FUNCTION "PressureAi" : VOID	// FC 29
TITLE = Block for pressure analog input
//Building:
//Date         Editor                                                     Version
//--------------------------------------------------------------------------------
//10.05.2017   (gea)                                                      01.00.00
//
//Modifications:
//No. Date     Edit  Description                                    Index Version
//--------------------------------------------------------------------------------
//01  
//________________________________________________________________________________
//Functional description:
//
//The Pressure Analogue Input Object includes the following functions
//- Check of overflow with substitude value
//- scaling of input value
//- check of pressure levels
//- mode selection 
//  manual mode (empty / convey / overpressure | zero pint adjustment)
//- overpressure detection (with delay)
//- overpressure alarm (with delay)
//- empty pressure detection (with delay)
//- active pressure detection 
//- adjustment of zeropoint (autoamtic / manual)
//- data structure for HMI connection
//
AUTHOR : gea
VERSION : 1.0
VAR_INPUT
  ManOpEn : BOOL ;	// Enable Manual mode
  ManModeTrack : BOOL ;	// Manual mode PV tracking
  NegEvalEn : BOOL ;	// overpressure=0; underpressure=1
  OVErrEn : BOOL ;	// overflow/underflow/broken wire error enable
  AlarmOprEn : BOOL ;	// Alarm high enable
  AlarmOprAckEn : BOOL ;	// Alarm high acknowledge enable
  DigitMin : INT ;	// scaling digit max
  DigitMax : INT ;	// scaling digit min
  ValueMin : REAL ;	// scaling value max
  ValueMax : REAL ;	// scaling value min
  ValueSubs : REAL ;	// substitude value
  Configuration : WORD ;	// external Configuration (0=use internal)
  UOM : INT ;	// external Uom  (0=use internal)
  iSystemOn : BOOL ;	// System activated
  iwDigit : INT ;	// input digit value
  iActive : BOOL ;	// Pressure montioring active
  aAlarmOprAck : BOOL ;	// Alarm high acknowledge
END_VAR
VAR_IN_OUT
  PVAct : REAL ;
  fAlarmOpr : BOOL ;
  OverPressure : BOOL ;
  EmptyPressure : BOOL ;
  ActivePressure : BOOL ;
  fScalingErr : BOOL ;
  fOVErr : BOOL ;
  fParErr : BOOL ;
  ioStructure : ANY ;
END_VAR
VAR_TEMP
  State : INT ;
  tempReal1 : REAL ;
  tempReal2 : REAL ;
  tempDB : INT ;
  PVActRaw : REAL ;
  ScaleingErrPV : BOOL ;
  ScaleingErrOffset : BOOL ;
END_VAR
BEGIN
NETWORK
TITLE =  get start byte of structure
      L     P##ioStructure;
      LAR2;
      L     W [AR2,P#4.0];
      T     #tempDB;
      OPN   DI [#tempDB];
      L     D [AR2,P#6.0];
      LAR2;
NETWORK
TITLE =  external  configuration
      L     #Configuration;
      L     0;
      ==I;
      JC    NECO;
      L     #Configuration;
      L     0;
      <>I;
      =     DIX [AR2,P#0.0];	// PressureAinOn
      L     #Configuration;
      L     2#1000;
      AW;
      L     0;
      <>I;
      =     DIX [AR2,P#0.3];	// counter overpressure on
      L     #Configuration;
      L     2#10000;
      AW;
      L     0;
      <>I;
      =     DIX [AR2,P#0.4];	// counter emptypressure on
      L     #Configuration;
      L     2#100000;
      AW;
      L     0;
      <>I;
      =     DIX [AR2,P#0.5];	// counter activepressure on
      L     #Configuration;
      L     2#100000000;
      AW;
      L     0;
      <>I;
      =     DIX [AR2,P#1.0];	// overpressure parameter on
      L     #Configuration;
      L     2#1000000000;
      AW;
      L     0;
      <>I;
      =     DIX [AR2,P#1.1];	// emptypressure parameter on
      L     #Configuration;
      L     2#10000000000;
      AW;
      L     0;
      <>I;
      =     DIX [AR2,P#1.2];	// activeypressure parameter on
      L     #Configuration;
      L     2#1000000000000;
      AW;
      L     0;
      <>I;
      =     DIX [AR2,P#1.4];	// manual operation simulation on
      L     #Configuration;
      L     2#10000000000000;
      AW;
      L     0;
      <>I;
      =     DIX [AR2,P#1.5];	// manual operation adjust on
NECO: NOP   0;
      L     #UOM;
      L     0;
      ==I;
      JC    NEUO;
      L     #UOM;
      T     DIW [AR2,P#2.0];
NEUO: NOP   0;
NETWORK
TITLE =  clean up configuration
      O     DIX [AR2,P#0.3];	// counter overpressure on
      R     DIX [AR2,P#0.4];	// counter emptypressure on
      O     DIX [AR2,P#0.3];	// counter overpressure on
      O     DIX [AR2,P#0.4];	// counter emptypressure on
      R     DIX [AR2,P#0.5];	// counter activepressure on
NETWORK
TITLE =  selection manual mode
      A     DIX [AR2,P#4.1];	// ManModeOp
      AN    DIX [AR2,P#4.2];	// ManModeLock
      AN    "M0.0 LockManualMode";	// manual mode general disabled
      S     DIX [AR2,P#4.0];	// ManModAct
      ON    DIX [AR2,P#4.1];	// ManModeOp
      ON    #ManOpEn;	// manual mode local disabled
      O     "M0.0 LockManualMode";	// manual mode general disabled
      O     DIX [AR2,P#4.2];	// ManModeLock
      R     DIX [AR2,P#4.0];	// ManModAct
      R     DIX [AR2,P#4.1];	// ManModeOp
NETWORK
TITLE =  overflow / underflow / broken wire check
      O(;
      L     #iwDigit;
      L     32511;
      >I;
      );	//overflow
      O(;
      A(;
      L     #iwDigit;
      L     -32512;
      <I;
      );
      A(;
      L     #DigitMin;
      L     0;
      <>I;	//bipolar
      );
      );	//underflow bipolar
      O(;
      A(;
      L     #iwDigit;
      L     -4864;
      <I;
      );
      A(;
      L     #DigitMin;
      L     0;
      ==I;	//unipolar
      );
      );	//underflow //unipolar
      A     #OVErrEn;	//enable overflow / underflow error
      =     #fOVErr;
NETWORK
TITLE =  scaling of PV
//Val = ValueMin + (ValueMax-ValueMin)*(iwDigit-DigitMin)/(DigitMax-DigitMin)
// (network holds code this reader does not know; not shown)
NETWORK
TITLE =  substidue PV
      O     #fScalingErr;
      O     #fOVErr;
      AN    DIX [AR2,P#4.0];	// ManModAct
      JCN   PVSU;
      L     #ValueSubs;
      T     #PVAct;
PVSU: NOP   0;
NETWORK
TITLE =  manual mode PV: off
      A     DIX [AR2,P#4.0];	// ManModAct
      AN    DIX [AR2,P#4.3];	// ManOpPressureEmpty
      AN    DIX [AR2,P#4.4];	// ManOpPressureConveying
      AN    DIX [AR2,P#4.5];	// ManOpPressureAlarm
      A     DIX [AR2,P#1.4];	// ManOpSimEn
      JCN   PVMO;
      L     0.000000e+00;
      T     #PVAct;
PVMO: NOP   0;
NETWORK
TITLE =  manual mode PV: Emptypressure
      A     DIX [AR2,P#4.0];	// ManModAct
      A     DIX [AR2,P#4.3];	// ManOpPressureEmpty
      AN    DIX [AR2,P#4.4];	// ManOpPressureConveying
      AN    DIX [AR2,P#4.5];	// ManOpPressureAlarm
      A     DIX [AR2,P#1.4];	// ManOpSimEn
      JCN   PVME;
      L     DID [AR2,P#24.0];	//EmptypressurePV     
      L     DID [AR2,P#28.0];	//ActivePressurePV    
      -R;
      L     2.000000e+00;
      /R;
      L     DID [AR2,P#28.0];	//ActivePressurePV    
      +R;
      T     #PVAct;
PVME: NOP   0;
NETWORK
TITLE =  manual mode PV: convey pressure
      A     DIX [AR2,P#4.0];	// ManModAct
      A     DIX [AR2,P#4.4];	// ManOpPressureConveying
      AN    DIX [AR2,P#4.5];	// ManOpPressureAlarm
      A     DIX [AR2,P#1.4];	// ManOpSimEn
      JCN   PVMC;
      L     DID [AR2,P#16.0];	//MaxpressurePV     
      L     DID [AR2,P#24.0];	//EmptypressurePV     
      -R;
      L     2.000000e+00;
      /R;
      L     DID [AR2,P#24.0];	//EmptypressurePV     
      +R;
      T     #PVAct;
PVMC: NOP   0;
NETWORK
TITLE =  manual mode PV: overpressure
      A     DIX [AR2,P#4.0];	// ManModAct
      A     DIX [AR2,P#4.5];	// ManOpPressureAlarm
      A     DIX [AR2,P#1.4];	// ManOpSimEn
      JCN   PVMA;
      L     DID [AR2,P#16.0];	//MaxpressurePV     
      T     #PVAct;
PVMA: NOP   0;
NETWORK
TITLE =  check Parameter
// (network holds code this reader does not know; not shown)
NETWORK
TITLE =  overpressure detection
      A(;
      L     #PVAct;
      L     DID [AR2,P#16.0];	//MaxpressurePV     
      >=R;
      );
      AN    #NegEvalEn;
      A     #iActive;
      O;
      A(;
      L     #PVAct;
      L     DID [AR2,P#16.0];	//MaxpressurePV     
      <=R;
      );
      A     #NegEvalEn;
      A     #iActive;
      S     #OverPressure;
      A(;
      L     #PVAct;
      L     DID [AR2,P#20.0];	//MinpressurePV 
      <=R;
      );
      AN    #NegEvalEn;
      O;
      A(;
      L     #PVAct;
      L     DID [AR2,P#20.0];	//MinpressurePV 
      >=R;
      );
      A     #NegEvalEn;
      ON    #iActive;
      R     #OverPressure;
NETWORK
TITLE =  emptypressure detection
      A(;
      L     #PVAct;
      L     DID [AR2,P#24.0];	//EmptypressurePV     
      <=R;
      );
      AN    #NegEvalEn;
      A     #iActive;
      O;
      A(;
      L     #PVAct;
      L     DID [AR2,P#24.0];	//EmptypressurePV     
      >=R;
      );
      A     #NegEvalEn;
      A     #iActive;
      JCN   EPDC;
      A     "M4.5 ImpulseClock1,0Sec";
      AN    #EmptyPressure;
      L     DIW [AR2,P#38.0];	// EmptyDelayCounter
      JCN   EPDR;
      +     1;
      JU    EPDR;
EPDC: L     0;
EPDR: T     DIW [AR2,P#38.0];	// EmptyDelayCounter
      L     DIW [AR2,P#32.0];	// EmptyDelay
      >=I;
      =     #EmptyPressure;
NETWORK
TITLE =  activepressure detection
      A(;
      L     #PVAct;
      L     DID [AR2,P#28.0];	//ActivePressurePV    
      >=R;
      );
      A     #iActive;
      AN    #NegEvalEn;
      O;
      A(;
      L     #PVAct;
      L     DID [AR2,P#28.0];	//ActivePressurePV    
      <=R;
      );
      A     #iActive;
      A     #NegEvalEn;
      JCN   APDC;
      A     "M4.5 ImpulseClock1,0Sec";
      AN    #ActivePressure;
      L     DIW [AR2,P#40.0];	// ActiveDelayCounter
      JCN   APDR;
      +     1;
      JU    APDR;
APDC: L     0;
APDR: T     DIW [AR2,P#40.0];	// ActiveDelayCounter
      L     DIW [AR2,P#34.0];	// ActiveDelay
      >=I;
      =     #ActivePressure;
NETWORK
TITLE =  Alarm overpressure
      A     #OverPressure;
      A     #AlarmOprEn;
      A     #iActive;
      JCN   OPDC;
      A     "M4.5 ImpulseClock1,0Sec";
      AN    #fAlarmOpr;
      L     DIW [AR2,P#42.0];	// AlarmDelayCounter
      JCN   OPDR;
      +     1;
      JU    OPDR;
OPDC: L     0;
OPDR: T     DIW [AR2,P#42.0];	// AlarmDelayCounter
      L     DIW [AR2,P#36.0];	// AlarmDelay
      >=I;
      S     #fAlarmOpr;
      AN    #OverPressure;
      A(;
      A     #AlarmOprAckEn;
      A     #aAlarmOprAck;
      ON    #AlarmOprAckEn;
      );
      ON    #AlarmOprEn;
      ON    #iSystemOn;
      ON    #iActive;
      R     #fAlarmOpr;
NETWORK
TITLE =  adjust automatic
// (network holds code this reader does not know; not shown)
NETWORK
TITLE =  adjust manual
      AN    DIX [AR2,P#4.0];	// ManModeAct
      A     DIX [AR2,P#1.5];	// parameter.MapOpAdjustEn
      A     DIX [AR2,P#4.6];	// ManOpPressureAdjust
      =     DIX [AR2,P#6.4];	// ManAdjustReq
      A     DIX [AR2,P#1.5];	// parameter.MapOpAdjustEn
      A     DIX [AR2,P#4.6];	// ManOpPressureAdjust
      AN    #iActive;
      A     DIX [AR2,P#6.4];	// ManAdjustReq
      A     DIX [AR2,P#6.5];	// ManAdjustRdy
      JCN   ADMA;
      L     #PVActRaw;
      T     DID [AR2,P#12.0];	//PressureOffset
      SET;	// done!
      R     DIX [AR2,P#4.6];	// ManOpPressureAdjust
ADMA: NOP   0;
      ON    DIX [AR2,P#1.5];	// parameter.MapOpAdjustEn
      R     DIX [AR2,P#4.6];	// ManOpPressureAdjust
NETWORK
TITLE =  Switch counter count up
      A     #OverPressure;
      A     DIX [AR2,P#0.3];	// parameter.counterOverPressure
      O;
      A     #EmptyPressure;
      A     DIX [AR2,P#0.4];	// parameter.counterEmptyPressure
      O;
      A     #ActivePressure;
      A     DIX [AR2,P#0.5];	// parameter.counterActivePressure
      FP    DIX [AR2,P#6.7];	// Switch counter edge
      JCN   SCUP;
      L     1.000000e+00;
      L     DID [AR2,P#44.0];	// Switch counter
      +R;
      T     DID [AR2,P#44.0];	// Switch counter
SCUP: NOP   0;
NETWORK
TITLE =  Switch counter reset
      A     DIX [AR2,P#6.6];	// Switch counter Reset
      O;
      AN    DIX [AR2,P#0.3];	// parameter.counterOverPressure
      AN    DIX [AR2,P#0.5];	// parameter.counterEmptyPressure
      AN    DIX [AR2,P#0.4];	// parameter.counterActivePressure
      JCN   SCRE;
      R     DIX [AR2,P#6.6];	// Switch counter Reset
      L     0.000000e+00;
      T     DID [AR2,P#44.0];	// Switch counter
SCRE: NOP   0;
NETWORK
TITLE =  track manual mode value in automatic
      AN    DIX [AR2,P#4.0];	// ManModAct
      A     #ManModeTrack;
      AN    #fParErr;
      JCN   PVTK;
      AN    #ActivePressure;
      AN    #EmptyPressure;
      AN    #OverPressure;
      R     DIX [AR2,P#4.3];	// ManOpPressureEmpty
      R     DIX [AR2,P#4.4];	// ManOpPressureConveying
      R     DIX [AR2,P#4.5];	// ManOpPressureAlarm
      A     #ActivePressure;
      A     #EmptyPressure;
      AN    #OverPressure;
      S     DIX [AR2,P#4.3];	// ManOpPressureEmpty
      R     DIX [AR2,P#4.4];	// ManOpPressureConveying
      R     DIX [AR2,P#4.5];	// ManOpPressureAlarm
      A     #ActivePressure;
      AN    #EmptyPressure;
      AN    #OverPressure;
      R     DIX [AR2,P#4.3];	// ManOpPressureEmpty
      S     DIX [AR2,P#4.4];	// ManOpPressureConveying
      R     DIX [AR2,P#4.5];	// ManOpPressureAlarm
      A     #ActivePressure;
      AN    #EmptyPressure;
      A     #OverPressure;
      R     DIX [AR2,P#4.3];	// ManOpPressureEmpty
      R     DIX [AR2,P#4.4];	// ManOpPressureConveying
      S     DIX [AR2,P#4.5];	// ManOpPressureAlarm
PVTK: NOP   0;
NETWORK
TITLE =  Objektstatus für Visualisation OP (009) (010)
// 9 = scaling/overflow/underflow/broken wire: substitude value ==> grey 
      L     9;
      O     #fScalingErr;
      O     #fOVErr;
      JC    disp;
// 19 = system not on (interlock) ==> orange
      L     19;
      AN    #iSystemOn;
      JC    disp;
// 16 = alarm overpressure ==> red
      L     16;
      A     #fAlarmOpr;
      JC    disp;
// 16 = overpressure ==> yellow
      L     13;
      A     #OverPressure;
      AN    #fAlarmOpr;
      JC    disp;
// 5 = switch on ==> green
      L     5;
      A     #ActivePressure;
      AN    #EmptyPressure;
      JC    disp;
// 1 = switch off ==> cyan
      L     1;
      A     #ActivePressure;
      A     #EmptyPressure;
      JC    disp;
      L     0;
disp: T     #State;
NETWORK
TITLE =  save data to structure
      A     #iSystemOn;
      =     DIX [AR2,P#4.7];
      A     #fScalingErr;
      =     DIX [AR2,P#5.0];
      A     #fOVErr;
      =     DIX [AR2,P#5.1];
      A     #fParErr;
      =     DIX [AR2,P#5.2];
      A     #fAlarmOpr;
      =     DIX [AR2,P#5.3];
      A     #AlarmOprEn;
      =     DIX [AR2,P#5.4];
      A     #aAlarmOprAck;
      =     DIX [AR2,P#5.5];
      A     #OverPressure;
      =     DIX [AR2,P#5.6];
      A     #EmptyPressure;
      =     DIX [AR2,P#5.7];
      A     #ActivePressure;
      =     DIX [AR2,P#6.0];
      A     #iActive;
      =     DIX [AR2,P#6.1];
      L     #PVAct;
      T     DID [AR2,P#8.0];
      L     #State;
      T     DIW [AR2,P#48.0];	// #Objektstatus  (Struktur) 
END_FUNCTION

FUNCTION "FC30 DB vorbelegen" : VOID	// FC 30
TITLE = Baustein vorbelegen
//Erstellung:
//Datum        Bearbeiter                                                 Version
//--------------------------------------------------------------------------------
//08.12.98     R.Schaffert (sra)                                          01.00.00
//
//Änderungen:
//Nr. Datum    Bearb Beschreibung                                   Marke Version
//--------------------------------------------------------------------------------
//01  13.04.00 sra   Fehlerbehebung (1 Byte zuviel belegt)                01.00.01
//02  25.08.00 sra   Fehlerbehebung Zeigerberechnung                      01.00.02
//
//________________________________________________________________________________
//Beschreibung:
//
//Diese Funktion beschreibt die angegebenen Worte eines Datenbausteins mit dem im 
//Parameter "Wert" eingetragenen Wert.
//
AUTHOR : sra
FAMILY : AZO
VERSION : 0.0
VAR_INPUT
  DB_Nr : INT ;	//Datenbausteinnummer
  DW_Anfang : INT ;	//Anfangs-Datenwort im Datenbaustein
  Anzahl_Bytes : INT ;	//Anzahl der Bytes die vorbelegt werden sollen
  Wert : INT ;	//Wert mit dem der Bereich vorbelegt werden soll
END_VAR
VAR_TEMP
  Datenbaustein : INT ;
  Ptr_aktuelles_Datenbyte : DWORD ;
  Ptr_Ende_Datenbyte : DWORD ;
END_VAR
BEGIN
NETWORK
TITLE = Anzahl Worte prüfen
      L     #Anzahl_Bytes;
      L     0;
      <=I;
      JC    Ende;
NETWORK
TITLE = Datenbaustein öffnen
      L     #DB_Nr;
      T     #Datenbaustein;
      OPN   DB [#Datenbaustein];
NETWORK
TITLE = Pointer belegen
      L     #DW_Anfang;
      SLD   3;
      T     #Ptr_aktuelles_Datenbyte;
      L     #Anzahl_Bytes;
      L     #DW_Anfang;
      +I;
      SLD   3;
      T     #Ptr_Ende_Datenbyte;
NETWORK
TITLE = Wert schreiben
Loop: NOP   0;
      L     #Wert;
      T     DBB [#Ptr_aktuelles_Datenbyte];
      L     #Ptr_aktuelles_Datenbyte;	// Wortadresse um 1 erhöhen
      L     P#1.0;
      +D;
      T     #Ptr_aktuelles_Datenbyte;
      L     #Ptr_Ende_Datenbyte;
      <D;
      JC    Loop;
Ende: NOP   0;
END_FUNCTION

FUNCTION "FC40 copy Obj-SST Master" : VOID	// FC 40
TITLE = SST an Slave
//Erstellung:
//Datum        Bearbeiter                                                 Version
//--------------------------------------------------------------------------------
//22.03.01     R.Schaffert (sra)                                          01.00.00
//
//Änderungen:
//Nr. Datum    Bearb Beschreibung                                   Marke Version
//--------------------------------------------------------------------------------
//01  16.08.01 sra   Fehlerbeseitigung  Daten löschen               (001) 01.00.01
//02  31.08.01 sra   Daten von Ziel auch löschen wenn Ziel-DB 0 ist (002) 01.00.02
//
//________________________________________________________________________________
//Beschreibung: 
//
//Der Baustein kopiert die Schnittstelle, die durch den ANY-Zeiger festgelegt 
//ist, 
//an einen "Slave". Sobald ein Bit in der Steuerbitleiste gesetzt ist reagiert 
//der 
//Slave und antwortet. Ist kein Bit in der Steuerbitleiste belegt, baut der Slave 
//die Schnittstelle ab und kann durch anderen Master belegt werden.
//!!Die Steuerbitleiste ist immer das letzte Wort in der Schnittstelle!!
//
//Anwendung z.B. bei Kommunikation mehrere Waage <-> mehrere Silo  
// 
//
AUTHOR : sra
FAMILY : AZO
VERSION : 0.0
VAR_INPUT
  i_Freigabe : BOOL ;	//Freigabe der Kopierfunktion
  i_Ziel_DB : INT ;	//Ziel-Datenbaustein
  i_Ziel_DW : INT ;	//Ziel-Datenwort im Ziel-Datenbaustein
  i_SST_von_Ziel : ANY ;	//ANY-Zeiger auf Schnittstellen von Slave
  i_SST_an_Ziel : ANY ;	//ANY-Zeiger auf Schnittstellen an Slave
END_VAR
VAR_OUTPUT
  Ziel_frei : BOOL ;	//"Slave" ist nicht durch anderen Master belegt,die Daten können umkopiert werden
END_VAR
VAR_TEMP
  Quell_DB : INT ;
  SST_an_Anfangs_DW : INT ;
  SST_an_Laenge : INT ;
  SST_von_Anfangs_DW : INT ;
  SST_von_Laenge : INT ;
  Ziel_DB : INT ;
  Zaehler : INT ;
  Fehler_Blockkopieren : INT ;
END_VAR
BEGIN
NETWORK
TITLE = ANY Zeiger "SST_von_Ziel" zerlegen
      L     P##i_SST_von_Ziel;
      LAR2;
      L     W [AR2,P#2.0];
      T     #SST_von_Laenge;
      L     D [AR2,P#6.0];
      L     DW#16#FFFFFF;
      AD;
      SRD   3;
      T     #SST_von_Anfangs_DW;
NETWORK
TITLE = ANY Zeiger "SST_an_Ziel" zerlegen
      L     P##i_SST_an_Ziel;
      LAR2;
      L     W [AR2,P#2.0];
      T     #SST_an_Laenge;
      L     W [AR2,P#4.0];
      T     #Quell_DB;
      L     D [AR2,P#6.0];
      L     DW#16#FFFFFF;
      AD;
      SRD   3;
      T     #SST_an_Anfangs_DW;
NETWORK
TITLE = Prüfen ob Ziel-DB <> 0
      L     #i_Ziel_DB;
      L     0;
      ==I;
      JC    DEL1;	// 002
NETWORK
TITLE = Prüfen ob Slave belegt ist
      L     #i_Ziel_DB;
      T     #Ziel_DB;
      OPN   DB [#Ziel_DB];
      L     #i_Ziel_DW;
      SLD   3;
      LAR2;
      O(;	// Slave bereits belegt ?
      L     DBW [AR2,P#0.0];
      L     #Quell_DB;
      ==I;
      );
      O(;	// Slave frei ?
      L     DBW [AR2,P#0.0];
      L     0;
      ==I;
      );
      =     #Ziel_frei;
NETWORK
TITLE = Daten von Ziel löschen
DEL1: OPN   DB [#Quell_DB];
      L     #SST_von_Anfangs_DW;
      SLD   3;
      LAR2;
      L     #SST_von_Laenge;
DEL2: T     #Zaehler;
      L     0;
      T     DBB [AR2,P#0.0];
      L     P#1.0;	// (001)
      +AR2;	// (001)
      L     #Zaehler;
      LOOP  DEL2;
      ON    #i_Freigabe;
      ON    #Ziel_frei;
      O(;	// (002)
      L     #i_Ziel_DB;	// (002)
      L     0;	// (002)
      ==I;	// (002)
      );	// (002)
      BEC;
NETWORK
TITLE = Daten an Slave kopieren
      L     #SST_an_Anfangs_DW;
      SLD   3;
      LAR2;
      L     #Quell_DB;
      T     DBW [AR2,P#0.0];
      L     #SST_von_Anfangs_DW;
      T     DBW [AR2,P#2.0];
      CALL  "FC5 Blocktransfer" (
           Quell_Typ                := B#16#44,
           Quell_DB                 := #Quell_DB,
           Quell_DW                 := #SST_an_Anfangs_DW,
           Ziel_Typ                 := B#16#44,
           Ziel_DB                  := #i_Ziel_DB,
           Ziel_DW                  := #i_Ziel_DW,
           Block_Laenge             := #SST_an_Laenge,
           outFehler                := #Fehler_Blockkopieren);
END_FUNCTION

FUNCTION "FC41 copy Obj-SST Slave" : VOID	// FC 41
TITLE = SST an Master
//Erstellung:
//Datum        Bearbeiter                                                 Version
//--------------------------------------------------------------------------------
//22.03.01     R.Schaffert (sra)                                          01.00.00
//
//Änderungen:
//Nr. Datum    Bearb Beschreibung                                   Marke Version
//--------------------------------------------------------------------------------
//01  00.00.00 xxx   xxx                                            ???   01.xx.xx
//
//________________________________________________________________________________
//Beschreibung: 
//
//Der Baustein kopiert die Schnittstelle, die durch den ANY-Zeiger festgelegt 
//ist, an einen "Master". Sobald ein Bit in der Steuerbitleiste gesetzt ist 
//reagiert der Slave und antwortet. Ist kein Bit in der Steuerbitleiste belegt, 
//baut der Slave die Schnittstelle ab und kann durch anderen Master belegt werden.
//!!Die Steuerbitleiste ist immer das letzte Wort in der Schnittstelle!!
//
//Anwendung z.B. bei Kommunikation mehrere Waage <-> mehrere Silo  
// 
//
//
AUTHOR : sra
FAMILY : AZO
VERSION : 0.0
VAR_INPUT
  i_SST_von_Ziel : ANY ;	//ANY-Zeiger auf Schnittstelle von Master
  i_SST_an_Ziel : ANY ;	//ANY-Zeiger auf Schnittstelle an Master
END_VAR
VAR_TEMP
  SST_an_Anfangs_DW : INT ;
  SST_an_Laenge : INT ;
  SST_von_Anfangs_DW : INT ;
  SST_von_Laenge : INT ;
  Ptr_SST_von_Anfangs_DW : DWORD ;
  Ptr_SST_von_Steuerbits : DWORD ;	//Steuerbits = Anfangs-DW + Länge -2
  Quell_DB : INT ;
  Ziel_DB : INT ;
  Ziel_DW : INT ;
  Fehler_Blockkopieren : INT ;
END_VAR
BEGIN
NETWORK
TITLE = ANY Zeiger "SST_von_Ziel" zerlegen
      L     P##i_SST_von_Ziel;
      LAR2;
      L     W [AR2,P#2.0];	// Länge der Struktur
      T     #SST_von_Laenge;
      L     D [AR2,P#6.0];	// Anfangs-DW der Struktur
      L     DW#16#FFFFFF;
      AD;
      SRD   3;
      T     #SST_von_Anfangs_DW;
NETWORK
TITLE = ANY Zeiger "SST_an_Ziel" zerlegen
      L     P##i_SST_an_Ziel;
      LAR2;
      L     W [AR2,P#2.0];
      T     #SST_an_Laenge;
      L     W [AR2,P#4.0];
      T     #Quell_DB;
      L     D [AR2,P#6.0];
      L     DW#16#FFFFFF;
      AD;
      SRD   3;
      T     #SST_an_Anfangs_DW;
NETWORK
TITLE = Pointer bilden
      L     #SST_von_Anfangs_DW;
      SLD   3;
      T     #Ptr_SST_von_Anfangs_DW;
      L     #SST_von_Anfangs_DW;
      L     #SST_von_Laenge;
      +I;
      L     2;
      -I;
      SLD   3;
      T     #Ptr_SST_von_Steuerbits;
NETWORK
TITLE = Prüfen ob Anforderung vorhanden
      OPN   DB [#Quell_DB];
      O(;
      L     DBW [#Ptr_SST_von_Anfangs_DW];	// Ziel-DB
      L     0;
      ==I;
      );
      O(;
      L     DBW [#Ptr_SST_von_Steuerbits];	// Steuerbits
      L     0;
      ==I;
      );
      JC    DEL;
NETWORK
TITLE = Daten an Master kopieren
      LAR2  #Ptr_SST_von_Anfangs_DW;
      L     DBW [AR2,P#0.0];	// Ziel-DB aus Struktur "SST_von" ermitteln
      T     #Ziel_DB;
      L     DBW [AR2,P#2.0];	// Ziel-DW aus Struktur "SST_von" ermitteln
      T     #Ziel_DW;
      CALL  "FC5 Blocktransfer" (
           Quell_Typ                := B#16#44,
           Quell_DB                 := #Quell_DB,
           Quell_DW                 := #SST_an_Anfangs_DW,
           Ziel_Typ                 := B#16#44,
           Ziel_DB                  := #Ziel_DB,
           Ziel_DW                  := #Ziel_DW,
           Block_Laenge             := #SST_an_Laenge,
           outFehler                := #Fehler_Blockkopieren);
NETWORK
TITLE = Daten von Master löschen
DEL:  L     DBW [#Ptr_SST_von_Steuerbits];
      L     0;
      <>I;
      JC    DELS;
      L     0;
      T     DBW [#Ptr_SST_von_Anfangs_DW];
DELS: L     0;
      T     DBW [#Ptr_SST_von_Steuerbits];
END_FUNCTION

FUNCTION "FC47 Tabelle schreiben" : VOID	// FC 47
TITLE = Tabelle schreiben
//DATUM     BEARBEITER                                                    VERSION
//--------------------------------------------------------------------------------
//29.02.00  A. Geiger (gea)                                               01.00.00
//  
//Änderungen:
//Nr. Datum    Bearb Beschreibung                                   Marke Version
//--------------------------------------------------------------------------------
//01  30.08.00 gea   Neue Konzeption (Kopieren über Schleife)             02.00.00
//
//________________________________________________________________________________
//Beschreibung: 
//Datensatz in Tabelle schreiben
//
//Aufbau Tabelle:
//  Tabellen-DB: 
//               DBB0    ... DBB(n-1)  1.Zeile
//               DBB(n)  ... DBB(2n-1) 2.Zeile
//               DBB(2n) ... DBB(3n-1) 3.Zeile
//               usw.
//
//Die Anzahl der Spalten pro Zeile (n) ist abhängig von der Länge der "Quelle".
//Die "Quelle" muß ein ANY-Zeiger auf Bytes oder Stuct sein.
//eine Überprüfung auf Existenz und Länge des Tabellen-DBs wird durchgeführt.
//
AUTHOR : gea
FAMILY : AZO
VERSION : 0.0
VAR_INPUT
  in_Tabelle_DB : INT ;	//Tabellen-DB-Nr.
  in_Offset_DW : INT ;	//Offset erster Tabelleneintrag in Tabellen-DB
  in_Zeile_schreiben : INT ;	//Eintrag in Tabelle, der geschrieben werden soll
END_VAR
VAR_OUTPUT
  out_Fehler : INT ;	//Fehlerauswertung
END_VAR
VAR_IN_OUT
  io_Quelle : ANY ;	//Zeiger auf Quelldaten Block
END_VAR
VAR_TEMP
  G_DB_SAVE : INT ;	//Global-DB-Register
  I_DB_SAVE : INT ;	//Instanz-DB-Register
  Zeiger_Quelle : DWORD ;
  DB_Quelle : INT ;
  Zeiger_Ziel : DWORD ;
  DB_Ziel : INT ;
  Blocklaenge : INT ;
  Datentyp : BYTE ;
  Start_DBB : INT ;
END_VAR
BEGIN
NETWORK
TITLE = DB-Register sichern
      L     DBNO;
      T     #G_DB_SAVE;
      L     DINO;
      T     #I_DB_SAVE;
NETWORK
TITLE = ANY-Zeiger Quelle zerlegen
      L     P##io_Quelle;
      LAR1;
      L     B [AR1,P#1.0];
      T     #Datentyp;
      L     W [AR1,P#2.0];
      T     #Blocklaenge;
      L     W [AR1,P#4.0];
      T     #DB_Quelle;
      L     D [AR1,P#6.0];
      T     #Zeiger_Quelle;
NETWORK
TITLE = Blocklänge prüfen
      L     #Blocklaenge;
      L     0;
      <=I;
      JC    BLFE;	//Blocklänge Fehler
NETWORK
TITLE = Datentyp prüfen
      L     #Datentyp;
      L     2;	//Datentyp = Byte oder Struct
      ==I;
      JCN   DTFE;
NETWORK
TITLE = Start-DBB des gewählten Eintrags
      L     #in_Zeile_schreiben;
      L     1;
      -I;
      L     #Blocklaenge;
      *I;
      L     #in_Offset_DW;
      +I;
      T     #Start_DBB;	//Start des n-ten Eintrags
NETWORK
TITLE = Bereichszeiger Zielzeiger
      L     W#16#85;
      CAD;
      L     #Start_DBB;
      SLD   3;
      +D;
      T     #Zeiger_Ziel;
NETWORK
TITLE = Ziel-DB
      L     #in_Tabelle_DB;
      T     #DB_Ziel;
NETWORK
TITLE = DBs aufschlagen
      L     #DB_Quelle;
      L     0;
      <>I;
      JCN   QNDB;
      OPN   DB [#DB_Quelle];
      L     DBNO;
      L     0;
      <=I;
      JC    DBNX;	//Fehler DB existiert nicht
      L     #Zeiger_Quelle;
      SRW   3;	//Anfangsbyte
      L     #Blocklaenge;
      +I;
      L     DBLG;
      >I;
      JC    DBLF;	//Fehler DB Länge nicht ausreichend
      L     #Zeiger_Quelle;
      L     DW#16#FFFFFF;
      AD;
      L     W#16#84;
      CAD;
      +D;
      T     #Zeiger_Quelle;
QNDB: L     #DB_Ziel;
      L     0;
      <>I;
      JCN   ZNDB;
      OPN   DI [#DB_Ziel];
      L     DINO;
      L     0;
      <=I;
      JC    DBNX;	//Fehler DB existiert nicht
      L     #Start_DBB;
      L     #Blocklaenge;
      +I;
      L     DILG;
      >I;
      JC    DBLF;	//Fehler DB Länge nicht ausreichend
ZNDB: NOP   0;
NETWORK
TITLE = Bytes kopieren
//geschwindigkeitsopitmiert:
//- Schleifenzäehler bleibt in AKKU1 und AKKU2
//- Kopieren über Worte, letztes Byte (ungerade Bytezahl) separat.
// (network holds code this reader does not know; not shown)
NETWORK
TITLE = Fehlerauswertung
      L     0;	//kein Fehler
      JU    SEFE;	//  setze Fehlerausgang
      L     -1;	//Bereichszeiger Quelle falsch
      JU    SEFE;	//  setze Fehlerausgang
      L     -2;	//Bereichszeiger Ziel falsch
      JU    SEFE;	//  setze Fehlerausgang
BLFE: L     -3;	//Blocklänge falsch
      JU    SEFE;	//  setze Fehlerausgang
DBNX: L     -4;	//Datenbaustein nicht existent 
      JU    SEFE;	//  setze Fehlerausgang
DBLF: L     -5;	//Datenbaustein Längenfehler
      JU    SEFE;	//  setze Fehlerausgang
DTFE: L     -6;	//Fehler Datentyp in ANY-Zeiger
SEFE: T     #out_Fehler;
NETWORK
TITLE = DB-Register wiederherstellen
      OPN   DB [#G_DB_SAVE];
      OPN   DI [#I_DB_SAVE];
NETWORK
TITLE = BIE-Bit zuweisen
      L     #out_Fehler;
      L     0;
      ==I;
      SAVE;
END_FUNCTION

FUNCTION "FC104 Blocktransf. ANY-Z" : VOID	// FC 104
TITLE = BlockTransfer mit ANY-Zeiger als Ziel
//DATUM     BEARBEITER                                                    VERSION
//--------------------------------------------------------------------------------
//29.02.00  A. Geiger (gea)                                               01.00.00
//  
//Änderungen:
//Nr. Datum    Bearb Beschreibung                    Änderung       Marke Version
//--------------------------------------------------------------------------------
//01  06.07.00 gea   Neue Konzeption (Kopieren über Schleife)             02.00.00
//02  26.10.01 gea   Fehlerbehebung DB überprüfen                   (002) 02.00.01
//03  05.11.03 gea   Alle Datentypen zulassen                       (003) 02.00.02
//04  10.06.10 sra   Bereich > 32767 kopieren                       (004) 02.00.03
//________________________________________________________________________________
//
//Funktion:
//
//Beschreibung: Kopieren Quelle nach Ziel (ANY-Zeiger)
//
//Datentyp:
//  P - Peripherie
//  E - Eingänge
//  A - Ausgänge
//  M - Merker
//  D - Datenbaustein in Quell_DB bzw. Ziel_DB
//  I - Instanz-DB in DI-Register
//  G - Global-DB in DB-Register
//  L - Lokaldaten
//  K - Bausteinvorbelegen mit Konstante in Quell_DW (Low-Byte) (nur für Quelle)
//
//
//
//
//
//
//
//
//
//
//
//
//
//THE HORROR CONTINUES ...
AUTHOR : gea
VERSION : 0.0
VAR_INPUT
  in_Quell_Typ : CHAR ;
  in_Quell_DB : INT ;	//Ziel-DB bei DW-Transfer
  in_Quell_DW : INT ;	//Byte-Adresse der Quelle
  in_Ziel : ANY ;
END_VAR
VAR_OUTPUT
  out_Fehler : INT ;	//Fehlermeldung
END_VAR
VAR_TEMP
  G_DB_SAVE : INT ;	//Global-DB-Register
  I_DB_SAVE : INT ;	//Instanz-DB-Register
  Zeiger_Quelle : DWORD ;
  DB_Quelle : INT ;
  Zeiger_Ziel : DWORD ;
  DB_Ziel : INT ;
  Blocklaenge : INT ;
  Datentyp : BYTE ;
END_VAR
BEGIN
NETWORK
TITLE = DB-Register sichern
      L     DBNO;
      T     #G_DB_SAVE;
      L     DINO;
      T     #I_DB_SAVE;
NETWORK
TITLE = ANY-Zeiger Ziel zerlegen
      L     P##in_Ziel;
      LAR1;
      L     B [AR1,P#1.0];
      T     #Datentyp;
      L     W [AR1,P#2.0];
      T     #Blocklaenge;
      L     W [AR1,P#4.0];
      T     #DB_Ziel;
      L     D [AR1,P#6.0];
      T     #Zeiger_Ziel;
NETWORK
TITLE = Blocklänge prüfen
      L     #Blocklaenge;
      L     0;
      <=I;
      JC    BLFE;	//Blocklänge Fehler
NETWORK
TITLE = Datentyp prüfen
      L     #Datentyp;
      L     0;	//Datentyp = Byte oder Struct //(003)
      <>I;
      JCN   DTFE;
NETWORK
TITLE = Bereichskennung Quellzeiger
      L     #in_Quell_Typ;
      L     'P';
      ==I;
      L     W#16#80;
      JC    BEKQ;
      L     #in_Quell_Typ;
      L     'E';
      ==I;
      L     W#16#81;
      JC    BEKQ;
      L     #in_Quell_Typ;
      L     'A';
      ==I;
      L     W#16#82;
      JC    BEKQ;
      L     #in_Quell_Typ;
      L     'M';
      ==I;
      L     W#16#83;
      JC    BEKQ;
      L     #in_Quell_Typ;
      L     'D';
      ==I;
      L     W#16#84;
      JC    BEKQ;
      L     #in_Quell_Typ;
      L     'I';
      ==I;
      L     W#16#84;
      JC    BEKQ;
      L     #in_Quell_Typ;
      L     'G';
      ==I;
      L     W#16#84;
      JC    BEKQ;
      L     #in_Quell_Typ;
      L     'L';
      ==I;
      L     W#16#87;
      JC    BEKQ;
      L     #in_Quell_Typ;
      L     'K';
      ==I;
      L     L#0;
      JC    BEK1;
      JU    BEFQ;	//Bereichskennung falsch Quelle
BEKQ: CAD;
      L     #in_Quell_DW;
      SLD   3;
      +D;
BEK1: T     #Zeiger_Quelle;
NETWORK
TITLE = Quell-DB
      L     #in_Quell_Typ;
      L     'D';
      ==I;
      L     #in_Quell_DB;
      JC    DBQ;
      L     #in_Quell_Typ;
      L     'I';
      ==I;
      L     DINO;
      JC    DBQ;
      L     #in_Quell_Typ;
      L     'G';
      ==I;
      L     DBNO;
      JC    DBQ;
      L     0;
DBQ:  T     #DB_Quelle;
NETWORK
TITLE = DBs aufschlagen
      O(;	//(002)
      L     #in_Quell_Typ;	//(002)
      L     'D';	//(002)
      ==I;	//(002)
      );	//(002)
      O(;	//(002)
      L     #in_Quell_Typ;	//(002)
      L     'I';	//(002)
      ==I;	//(002)
      );	//(002)
      O(;	//(002)
      L     #in_Quell_Typ;	//(002)
      L     'G';	//(002)
      ==I;	//(002)
      );	//(002)
      JCN   QNDB;
      OPN   DB [#DB_Quelle];
      L     DBNO;
      L     0;
      <=I;
      JC    DBNX;	//Fehler DB existiert nicht
      L     #in_Quell_DW;
      L     #Blocklaenge;
      +D;	// (004)
      L     DBLG;
      >D;	// (004)
      JC    DBLF;	//Fehler DB Länge nicht ausreichend
QNDB: L     #DB_Ziel;
      L     0;
      <>I;
      JCN   ZNDB;
      OPN   DI [#DB_Ziel];
      L     DINO;
      L     0;
      <=I;
      JC    DBNX;	//Fehler DB existiert nicht
      L     #Zeiger_Ziel;
      SRW   3;	//Anfangsbyte
      L     #Blocklaenge;
      +D;	// (004)
      L     DILG;
      >D;	// (004)
      JC    DBLF;	//Fehler DB Länge nicht ausreichend
      L     #Zeiger_Ziel;
      L     DW#16#FFFFFF;
      AD;
      L     W#16#85;
      CAD;
      +D;
      T     #Zeiger_Ziel;
ZNDB: NOP   0;
NETWORK
TITLE = Bereich vorbelegen
//geschwindigkeitsopitmiert:
//- Schleifenzäehler bleibt in AKKU1 und AKKU2
//- Kopieren über Worte, letztes Byte (ungerade Bytezahl) separat.
      L     #in_Quell_Typ;
      L     'K';
      ==I;
      JCN   NKCO;
      L     #Zeiger_Ziel;
      LAR2;
      L     #in_Quell_DW;	//Konstante für vorbelegen
      L     #in_Quell_DW;
      SLW   8;	//  In AKKU1LL und AKKU1LH
      OW;
      L     #Blocklaenge;	//Schleifenzähler Blocklaenge->AKKU1
      SRW   1;
SCHK: TAK;	//Schleifenzähler AKKU1->AKKU2; Vorbelegwert in AKKU1
      T     W [AR2,P#0.0];
      +AR2  P#2.0;
      TAK;	//Schleifenzähler in AKKU2->AKKU1; Vorbelegwert in AKKU2
      LOOP  SCHK;
      JZ    BLGK;	//Gerade Byteanzahl A1=0 und A0=0 nach "SRW 1"
      L     #in_Quell_DW;	//Ungerade Bytezahl letztes Byte einzeln Kopieren
      SRW   8;
      T     B [AR2,P#0.0];
BLGK: NOP   0;
      JU    BLGE;
NKCO: NOP   0;
NETWORK
TITLE = Bytes kopieren
//geschwindigkeitsopitmiert:
//- Schleifenzäehler bleibt in AKKU1 und AKKU2
//- Kopieren über Worte, letztes Byte (ungerade Bytezahl) separat.
// (network holds code this reader does not know; not shown)
NETWORK
TITLE = Fehlerauswertung
      L     0;	//kein Fehler
      JU    SEFE;	//  setze Fehlerausgang
BEFQ: L     -1;	//Bereichszeiger Quelle falsch
      JU    SEFE;	//  setze Fehlerausgang
      L     -2;	//Bereichszeiger Ziel falsch
      JU    SEFE;	//  setze Fehlerausgang
BLFE: L     -3;	//Blocklänge falsch
      JU    SEFE;	//  setze Fehlerausgang
DBNX: L     -4;	//Datenbaustein nicht existent 
      JU    SEFE;	//  setze Fehlerausgang
DBLF: L     -5;	//Datenbaustein Längenfehler
      JU    SEFE;	//  setze Fehlerausgang
DTFE: L     -6;	//Fehler Datentyp in ANY-Zeiger
SEFE: T     #out_Fehler;
NETWORK
TITLE = DB-Register wiederherstellen
      OPN   DB [#G_DB_SAVE];
      OPN   DI [#I_DB_SAVE];
NETWORK
TITLE = BIE-Bit zuweisen
      L     #out_Fehler;
      L     0;
      ==I;
      SAVE;
END_FUNCTION

FUNCTION "FC113 Standardsignale 2" : VOID	// FC 113
TITLE = function for several cabinets with their own fuse check
//Erstellung:
//Date        developer                                                  version
//--------------------------------------------------------------------------------
//18.07.2016  A.Kremer (kal)                                             01.00.00
//
//changes:
//No. Date    developer description                                 Mark  version
//--------------------------------------------------------------------------------
//
//________________________________________________________________________________
//function:
//function, if more than one cabinet handle their own fuse check.
//function can be called several times, then.
//
AUTHOR : kal
FAMILY : AZO
VERSION : 0.0
VAR_INPUT
  iFaultFuse_OK : BOOL ;	//Eingang Sicherung OK = Eingang Störung Sicherung
END_VAR
VAR_OUTPUT
  qlFaultFuse : BOOL ;	//Ausgang der Lampe "Störung Sicherung"
  qFaultFuse : BOOL ;	//Störung Sicherung -> für Störbitzuweisung im DB34
END_VAR
BEGIN
NETWORK
TITLE = lamp "fault fuse" and fault message
      AN    #iFaultFuse_OK;
      =     #qlFaultFuse;
      =     #qFaultFuse;
END_FUNCTION

FUNCTION "FC6079 SimAnalog" : INT	// FC 6079
TITLE = simulate analog signal
//creation:
//date         who                                                         version
//--------------------------------------------------------------------------------
//28.12.2010   M. Junker (jm)                                             01.00.00
//
//changes:
//no. date       who            what                                       version
//--------------------------------------------------------------------------------
// 1  
//
//Function:
//simulates a slow changing analog signal (pressure, temperature) for 
//visualization tests or program tests
//
//y = a * sin(x) + b
AUTHOR : jm
FAMILY : AZO
NAME : SIMUL
VERSION : 0.1
VAR_INPUT
  RELEASE : BOOL ;	//release simulation
  PERIOD : REAL ;	//period time for sin() [s]
  MAX : REAL ;	//maximum analog value to simulate
  MIN : REAL ;	//minimum analog value to simulate
  DEFAULT : REAL ;	//default value if not simulating
  MAXVALUE : REAL ;	//upper limit analog value
  MINVALUE : REAL ;	//lower limit analog value
END_VAR
VAR_OUTPUT
  RET_VAL : INT ;	//simulated analog signal
END_VAR
VAR_IN_OUT
  STARTTIME : TIME ;	//starttime [ms]
  ONESHOTSTART : BOOL ;	//help flag start
END_VAR
VAR_TEMP
  ACTTIME : TIME ;
  y : REAL ;
  x : REAL ;
  a : REAL ;
  b : REAL ;
  MR1 : REAL ;
  MR2 : REAL ;
END_VAR
BEGIN
NETWORK
TITLE = detect start time
      A     #RELEASE;
      FP    #ONESHOTSTART;
      JCN   NSST;	// Not Set Start Time
      CALL  "TIME_TCK" (
           RET_VAL                  := #STARTTIME);
NSST: NOP   0;
NETWORK
TITLE = check if simulation necessary
      A     #RELEASE;
      JC    CONT;
      L     #DEFAULT;
      T     #y;
      JU    OUT;	// scale value for output
NETWORK
TITLE = calculate x
//x = 2*pi/1000/PERIOD*deltaTms = deltaTms*pi/500/PERIOD
CONT: CALL  "TIME_TCK" (
           RET_VAL                  := #ACTTIME);
      L     #ACTTIME;
      L     #STARTTIME;
      -D;	// deltaT in ms 
      DTR;
      L     3.141593e+00;	// PI
      *R;
      L     5.000000e+02;
      /R;
      L     #PERIOD;
      /R;
      T     #x;
NETWORK
TITLE = calculate a
//a = (MAX-MIN)/2
      L     #MAX;
      L     #MIN;
      -R;
      L     2.000000e+00;
      /R;
      T     #a;
NETWORK
TITLE = calculate b
//b = (MAX+MIN)/2
      L     #MAX;
      L     #MIN;
      +R;
      L     2.000000e+00;
      /R;
      T     #b;
NETWORK
TITLE = calculate y
//y = a*sin(x)+b
// (network holds code this reader does not know; not shown)
NETWORK
TITLE = scale output
//z = (MAXDIGIT-MINDIGIT)/(MAXVALUE-MINVALUE)*(y-MINVALUE)+MINDIGIT 
OUT:  L     #MAXVALUE;
      L     #MINVALUE;
      -R;
      T     #MR1;
      L     #y;
      L     #MINVALUE;
      -R;
      T     #MR2;
      L     2.764800e+04;
      L     #MR1;
      /R;
      L     #MR2;
      *R;
      RND;
      T     #RET_VAL;
END_FUNCTION

FUNCTION "FC6091 SimValve3A3E" : VOID	// FC 6091
TITLE = simulate valve 3A3E
//creation:
//date         who                                                         version
//--------------------------------------------------------------------------------
//04.12.2015   M. Junker (jm)                                             01.00.00
//
//changes:
//no. date       who            what                                       version
//--------------------------------------------------------------------------------
// 1  
//
//Function:
//simulate valve
AUTHOR : jm
FAMILY : AZO
NAME : SIMUL
VERSION : 1.0
VAR_INPUT
  o_ValveOn : BOOL ;
  o_ValveOff : BOOL ;
  o_ValveSealup : BOOL ;
END_VAR
VAR_OUTPUT
  i_ValveOn : BOOL ;	//on, open, pos1, ...
  i_ValveOff : BOOL ;	//off, closed, pos2, ...
  i_ValveSealed : BOOL ;	//sealed
END_VAR
VAR_IN_OUT
  mPosition : BOOL ;	//help memory
END_VAR
BEGIN
NETWORK
TITLE = valve on
      A     #o_ValveOn;
      S     #mPosition;
NETWORK
TITLE = valve off
      A     #o_ValveOff;
      R     #mPosition;
NETWORK
TITLE = indications
      A     #mPosition;
      =     #i_ValveOn;
      NOT;
      =     #i_ValveOff;
NETWORK
TITLE = sealed
      A     #o_ValveSealup;
      =     #i_ValveSealed;
END_FUNCTION

FUNCTION "FC6092 SimValveDOS" : VOID	// FC 6092
TITLE = simulate valve 2A2E (dosing valve)
//creation:
//date         who                                                         version
//--------------------------------------------------------------------------------
//05.06.2014   M. Junker (jm)                                             01.00.00
//
//changes:
//no. date       who            what                                       version
//--------------------------------------------------------------------------------
// 1  
//
//Function:
//simulate valve
AUTHOR : jm
FAMILY : AZO
NAME : SIMUL
VERSION : 1.0
VAR_INPUT
  in_Ventil_Typ : INT ;	//siehe Funktionsbeschreibung unten
  o_ValveCoarse : BOOL ;
  o_ValveFine : BOOL ;
END_VAR
VAR_OUTPUT
  i_ValveOpen : BOOL ;	//on, open, pos1, ...
  i_ValveClosed : BOOL ;	//off, closed, pos2, ...
END_VAR
VAR_IN_OUT
  mPosition : BOOL ;	//help memory
END_VAR
BEGIN
NETWORK
TITLE = valve open
      A     #o_ValveCoarse;
      S     #mPosition;
NETWORK
TITLE = valve  closed
      AN    #o_ValveCoarse;
      AN    #o_ValveFine;
      R     #mPosition;
NETWORK
TITLE = valve type 0
      A(;
      L     #in_Ventil_Typ;
      L     0;
      );
      <>I;
      JC    NVT0;
      A     #o_ValveCoarse;
      =     #i_ValveOpen;
      AN    #o_ValveCoarse;
      AN    #o_ValveFine;
      =     #i_ValveClosed;
NVT0: NOP   0;
NETWORK
TITLE = valve type 1
      A(;
      L     #in_Ventil_Typ;
      L     1;
      );
      <>I;
      JC    NVT1;
      A     #mPosition;
      =     #i_ValveOpen;
      AN    #mPosition;
      =     #i_ValveClosed;
NVT1: NOP   0;
NETWORK
TITLE = valve type 2
      A(;
      L     #in_Ventil_Typ;
      L     2;
      );
      <>I;
      JC    NVT2;
      A     #mPosition;
      =     #i_ValveOpen;
      AN    #mPosition;
      =     #i_ValveClosed;
NVT2: NOP   0;
END_FUNCTION

FUNCTION "FC6093 SimValveDS" : VOID	// FC 6093
TITLE = simulate valve 2A2E (double seat)
//creation:
//date         who                                                         version
//--------------------------------------------------------------------------------
//27.05.2014   M. Junker (jm)                                             01.00.00
//
//changes:
//no. date       who            what                                       version
//--------------------------------------------------------------------------------
// 1  
//
//Function:
//simulate valve
AUTHOR : jm
FAMILY : AZO
NAME : SIMUL
VERSION : 1.0
VAR_INPUT
  o_Valve_E0 : BOOL ;
  o_Valve_E1 : BOOL ;
END_VAR
VAR_OUTPUT
  i_Valve_A0 : BOOL ;	//on, open, pos1, ...
  i_Valve_A1 : BOOL ;	//off, closed, pos2, ...
END_VAR
BEGIN
NETWORK
TITLE = valve open
      A     #o_Valve_E0;
      A     #o_Valve_E1;
      =     #i_Valve_A1;
NETWORK
TITLE = valve close
      ON    #o_Valve_E0;
      ON    #o_Valve_E1;
      =     #i_Valve_A0;
END_FUNCTION

FUNCTION "FC6094 SimMotor2A2E" : VOID	// FC 6094
TITLE = simulate motor 2A2E+iso
//creation:
//date         who                                                         version
//--------------------------------------------------------------------------------
//05.06.2014   M. Junker (jm)                                             01.00.00
//
//changes:
//no. date       who            what                                       version
//--------------------------------------------------------------------------------
// 1  
//
//Function:
//simulate motor + isolator
AUTHOR : jm
FAMILY : AZO
NAME : SIMUL
VERSION : 1.0
VAR_INPUT
  o_MotorCW : BOOL ;
  o_MotorACW : BOOL ;
  Isolators : BOOL ;
END_VAR
VAR_OUTPUT
  i_MotorCW : BOOL ;
  i_MotorACW : BOOL ;
  i_IsoMotor : BOOL ;
END_VAR
BEGIN
NETWORK
TITLE = motor CW
      A     #o_MotorCW;
      =     #i_MotorCW;
NETWORK
TITLE = motor ACW
      A     #o_MotorACW;
      =     #i_MotorACW;
NETWORK
TITLE = isolator
      A     #Isolators;
      =     #i_IsoMotor;
END_FUNCTION

FUNCTION "FC6095 SimValve2A2E" : VOID	// FC 6095
TITLE = simulate valve 2A2E
//creation:
//date         who                                                         version
//--------------------------------------------------------------------------------
//25.10.2010   M. Junker (jm)                                             01.00.00
//
//changes:
//no. date       who            what                                       version
//--------------------------------------------------------------------------------
// 1  
//
//Function:
//simulate valve
AUTHOR : jm
FAMILY : AZO
NAME : SIMUL
VERSION : 1.0
VAR_INPUT
  o_ValveOn : BOOL ;
  o_ValveOff : BOOL ;
END_VAR
VAR_OUTPUT
  i_ValveOn : BOOL ;	//on, open, pos1, ...
  i_ValveOff : BOOL ;	//off, closed, pos2, ...
END_VAR
VAR_IN_OUT
  mPosition : BOOL ;	//help memory
END_VAR
BEGIN
NETWORK
TITLE = valve on
      A     #o_ValveOn;
      S     #mPosition;
NETWORK
TITLE = valve off
      A     #o_ValveOff;
      R     #mPosition;
NETWORK
TITLE = indications
      A     #mPosition;
      =     #i_ValveOn;
      NOT;
      =     #i_ValveOff;
END_FUNCTION

FUNCTION "FC6096 SimValve1AE1" : VOID	// FC 6096
TITLE = simulate valve 1AE1
//creation:
//date         who                                                         version
//--------------------------------------------------------------------------------
//25.10.2010   M. Junker (jm)                                             01.00.00
//
//changes:
//no. date       who            what                                       version
//--------------------------------------------------------------------------------
// 1  
//
//Function:
//simulate valve
AUTHOR : jm
FAMILY : AZO
NAME : SIMUL
VERSION : 1.0
VAR_INPUT
  o_ValveOn : BOOL ;
END_VAR
VAR_OUTPUT
  i_ValveOff : BOOL ;	//off, closed, pos2, ...
END_VAR
BEGIN
NETWORK
TITLE = valve off
      AN    #o_ValveOn;
      =     #i_ValveOff;
END_FUNCTION

FUNCTION "FC6097 SimValve1A1E" : VOID	// FC 6097
TITLE = simulate valve 1A1E
//creation:
//date         who                                                         version
//--------------------------------------------------------------------------------
//25.10.2010   M. Junker (jm)                                             01.00.00
//
//changes:
//no. date       who            what                                       version
//--------------------------------------------------------------------------------
// 1  
//
//Function:
//simulate valve
AUTHOR : jm
FAMILY : AZO
NAME : SIMUL
VERSION : 1.0
VAR_INPUT
  o_ValveOn : BOOL ;
END_VAR
VAR_OUTPUT
  i_ValveOn : BOOL ;	//on, open, pos1, ...
END_VAR
BEGIN
NETWORK
TITLE = valve on
      A     #o_ValveOn;
      =     #i_ValveOn;
END_FUNCTION

FUNCTION "FC6098 SimValve1A2E" : VOID	// FC 6098
TITLE = simulate valve 1A2E
//creation:
//date         who                                                         version
//--------------------------------------------------------------------------------
//25.10.2010   M. Junker (jm)                                             01.00.00
//
//changes:
//no. date       who            what                                       version
//--------------------------------------------------------------------------------
// 1  
//
//Function:
//simulate valve
AUTHOR : jm
FAMILY : AZO
NAME : SIMUL
VERSION : 1.0
VAR_INPUT
  o_ValveOn : BOOL ;
END_VAR
VAR_OUTPUT
  i_ValveOn : BOOL ;	//on, open, pos1, ...
  i_ValveOff : BOOL ;	//off, closed, pos2, ...
END_VAR
BEGIN
NETWORK
TITLE = valve on
      A     #o_ValveOn;
      =     #i_ValveOn;
NETWORK
TITLE = valve off
      AN    #o_ValveOn;
      =     #i_ValveOff;
END_FUNCTION

FUNCTION "FC6099 SimMotor1A1E" : VOID	// FC 6099
TITLE = simulate motor 1A1E+iso
//creation:
//date         who                                                         version
//--------------------------------------------------------------------------------
//25.10.2010   M. Junker (jm)                                             01.00.00
//
//changes:
//no. date       who            what                                       version
//--------------------------------------------------------------------------------
// 1  
//
//Function:
//simulate motor + isolator
AUTHOR : jm
FAMILY : AZO
NAME : SIMUL
VERSION : 1.0
VAR_INPUT
  o_MotorOn : BOOL ;
  Isolators : BOOL ;
END_VAR
VAR_OUTPUT
  i_MotorOn : BOOL ;
  i_IsoMotor : BOOL ;
END_VAR
BEGIN
NETWORK
TITLE = motor
      A     #o_MotorOn;
      =     #i_MotorOn;
NETWORK
TITLE = isolator
      A     #Isolators;
      =     #i_IsoMotor;
END_FUNCTION

DATA_BLOCK "CMs_SIMULATION_DB"	// DB 2
VERSION : 0.0
"CMs_SIMULATION"
BEGIN
END_DATA_BLOCK

DATA_BLOCK "DB3 CPU Daten"	// DB 3
AUTHOR : sra
FAMILY : AZO
VERSION : 0.0
  STRUCT
   OB1_Info : STRUCT
    OB1_DATE_TIME : DATE_AND_TIME ;	//Date and time OB1 started
    OB1_PREV_CYCLE : INT ;	//Cycle time of previous OB1 scan (milliseconds)
    OB1_MIN_CYCLE : INT ;	//Minimum cycle time of OB1 (milliseconds)
    OB1_MAX_CYCLE : INT ;	//Maximum cycle time of OB1 (milliseconds)
    reserve : ARRAY  [0 .. 14 ] OF BYTE ;
   END_STRUCT ;
   Fehler_OB_Info : STRUCT
    Zeitfehler_OB80 : BOOL ;	//Zeitfehler OB 80
    Stromversorgung_OB81 : BOOL ;	//Stromversorgungsfehler OB 81
    Diagnose_Alarm_OB82 : BOOL ;	//Diagnose-Alarm OB82
    Ziehen_Stecken_OB83 : BOOL ;	//Ziehen/Stecken-Alarm OB83
    CPU_Hardware_OB84 : BOOL ;	//CPU-Hardwarefehler OB84
    Programmablauf_OB85 : BOOL ;	//Programmablauffehler OB85
    Baugr_tr_ausfall_OB86 : BOOL ;	//Baugruppenträgerausfall OB86
    Kommunikation_OB87 : BOOL ;	//Kommunikationsfehler OB87
    Programmierfehler_OB121 : BOOL ;	//Programmierfehler OB121
    Periphzugriff_OB122 : BOOL ;	//Peripheriezugriffsfehler OB 122
    Bearbeitungsabbruch_OB88 : BOOL ;	//Bearbeitungsabbruch eines Bausteins OB88
    Battery_fault : BOOL ;	//Battery fault with SFC51
    reserve_word : WORD ;
    OB_80_Fault_ID : BYTE ;	//Fehlercode OB 80
    OB_81_Fault_ID : BYTE ;	//Fehlercode OB 81
    OB_82_Fault_ID : BYTE ;	//Fehlercode OB 82
    OB_83_Fault_ID : BYTE ;	//Fehlercode OB 83
    OB_84_Fault_ID : BYTE ;	//Fehlercode OB 84
    OB_85_Fault_ID : BYTE ;	//Fehlercode OB 85
    OB_86_Fault_ID : BYTE ;	//Fehlercode OB 86
    OB_87_Fault_ID : BYTE ;	//Fehlercode OB 87
    OB_121_Fault_ID : BYTE ;	//Fehlercode OB 121
    OB_122_Fault_ID : BYTE ;	//Fehlercode OB 122
    OB_88_Fault_ID : BYTE ;	//Fehlercode OB 122
    reserve : ARRAY  [16 .. 29 ] OF BYTE ;
   END_STRUCT ;
   RDSYSST : STRUCT
    BUSY : BOOL ;
    RETVAL : INT ;
    SLZ_HEADER : STRUCT
     LENTHDR : WORD ;
     N_DR : WORD ;
    END_STRUCT ;
    DR : STRUCT
     Data_1 : BYTE ;
     Data_2 : BYTE ;
     Data_3 : BYTE ;
     Data_4 : BYTE ;
     Data_5 : BYTE ;
     Data_6 : BYTE ;
     Data_7 : BYTE ;
     Data_8 : BYTE ;
     Data_9 : BYTE ;
     Data_10 : BYTE ;
     Data_11 : BYTE ;
     Data_12 : BYTE ;
     Data_13 : BYTE ;
     Data_14 : BYTE ;
     Data_15 : BYTE ;
     Data_16 : BYTE ;
     Data_17 : BYTE ;
     Data_18 : BYTE ;
     Data_19 : BYTE ;
     Data_20 : BYTE ;
    END_STRUCT ;
   END_STRUCT ;
  END_STRUCT ;	
BEGIN
END_DATA_BLOCK

DATA_BLOCK "DB4 Motordaten für FUs"	// DB 4
VERSION : 0.1
  STRUCT
   Motordaten1 : STRUCT 	//Anzahl der Motordaten abhängig von der Anzahl der verschied. benutzten Motoren
    Nennleistungsfaktor : REAL  := 8.000000e-001;	//Motornennleistungsfaktor cos phi
    Nennfrequenz : REAL  := 5.100000e+001;	//Motornennfrequenz in Einheit Hz
    Nenndrehzahl : REAL  := 1.400000e+003;	//Motornenndrehzal in U/min
    Nennstrom : REAL  := 6.100000e+000;	//Motornennstrom in A
    Nennspannung : REAL  := 2.310000e+002;	//Motornennspannung in V
    Nennleistung : REAL  := 1.400000e+000;	//Motornennleistung kW
    reserve : ARRAY  [24 .. 29 ] OF //Reserve für weitere Motordaten
    BYTE ;
   END_STRUCT ;
   Motordaten2 : STRUCT
    Nennleistungsfaktor : REAL  := 7.000000e-001;
    Nennfrequenz : REAL  := 1.000000e+002;
    Nenndrehzahl : REAL  := 2.000000e+002;
    Nennstrom : REAL  := 2.000000e+000;
    Nennspannung : REAL  := 3.800000e+002;
    Nennleistung : REAL  := 1.000000e+003;
    reserve : ARRAY  [24 .. 29 ] OF BYTE ;
   END_STRUCT ;
   Motordaten3 : STRUCT
    Nennleistungsfaktor : REAL  := 7.000000e-001;
    Nennfrequenz : REAL  := 1.000000e+002;
    Nenndrehzahl : REAL  := 2.000000e+002;
    Nennstrom : REAL  := 5.000000e+000;
    Nennspannung : REAL  := 3.800000e+002;
    Nennleistung : REAL  := 1.000000e+003;
    reserve : ARRAY  [24 .. 29 ] OF BYTE ;
   END_STRUCT ;
   Motordaten4 : STRUCT
    Nennleistungsfaktor : REAL  := 7.000000e-001;
    Nennfrequenz : REAL  := 1.000000e+002;
    Nenndrehzahl : REAL  := 2.000000e+002;
    Nennstrom : REAL  := 5.000000e+000;
    Nennspannung : REAL  := 3.800000e+002;
    Nennleistung : REAL  := 1.000000e+003;
    reserve : ARRAY  [24 .. 29 ] OF BYTE ;
   END_STRUCT ;
   Motordaten5 : STRUCT
    Nennleistungsfaktor : REAL  := 7.000000e-001;
    Nennfrequenz : REAL  := 1.000000e+002;
    Nenndrehzahl : REAL  := 2.000000e+002;
    Nennstrom : REAL  := 5.000000e+000;
    Nennspannung : REAL  := 3.800000e+002;
    Nennleistung : REAL  := 1.000000e+003;
    reserve : ARRAY  [24 .. 29 ] OF BYTE ;
   END_STRUCT ;
   Motordaten6 : STRUCT
    Nennleistungsfaktor : REAL  := 7.000000e-001;
    Nennfrequenz : REAL  := 1.000000e+002;
    Nenndrehzahl : REAL  := 2.000000e+002;
    Nennstrom : REAL  := 5.000000e+000;
    Nennspannung : REAL  := 3.800000e+002;
    Nennleistung : REAL  := 1.000000e+003;
    reserve : ARRAY  [24 .. 29 ] OF BYTE ;
   END_STRUCT ;
   Motordaten7 : STRUCT
    Nennleistungsfaktor : REAL  := 7.000000e-001;
    Nennfrequenz : REAL  := 1.000000e+002;
    Nenndrehzahl : REAL  := 2.000000e+002;
    Nennstrom : REAL  := 5.000000e+000;
    Nennspannung : REAL  := 3.800000e+002;
    Nennleistung : REAL  := 1.000000e+003;
    reserve : ARRAY  [24 .. 29 ] OF BYTE ;
   END_STRUCT ;
   Motordaten8 : STRUCT
    Nennleistungsfaktor : REAL  := 7.000000e-001;
    Nennfrequenz : REAL  := 1.000000e+002;
    Nenndrehzahl : REAL  := 2.000000e+002;
    Nennstrom : REAL  := 5.000000e+000;
    Nennspannung : REAL  := 3.800000e+002;
    Nennleistung : REAL  := 1.000000e+003;
    reserve : ARRAY  [24 .. 29 ] OF BYTE ;
   END_STRUCT ;
   Motordaten9 : STRUCT
    Nennleistungsfaktor : REAL  := 7.000000e-001;
    Nennfrequenz : REAL  := 1.000000e+002;
    Nenndrehzahl : REAL  := 2.000000e+002;
    Nennstrom : REAL  := 5.000000e+000;
    Nennspannung : REAL  := 3.800000e+002;
    Nennleistung : REAL  := 1.000000e+003;
    reserve : ARRAY  [24 .. 29 ] OF BYTE ;
   END_STRUCT ;
   Motordaten10 : STRUCT
    Nennleistungsfaktor : REAL  := 7.000000e-001;
    Nennfrequenz : REAL  := 1.000000e+002;
    Nenndrehzahl : REAL  := 2.000000e+002;
    Nennstrom : REAL  := 5.000000e+000;
    Nennspannung : REAL  := 3.800000e+002;
    Nennleistung : REAL  := 1.000000e+003;
    reserve : ARRAY  [24 .. 29 ] OF BYTE ;
   END_STRUCT ;
  END_STRUCT ;	
BEGIN
   Motordaten1.Nennleistungsfaktor := 8.000000e-01;
   Motordaten1.Nennfrequenz := 5.100000e+01;
   Motordaten1.Nenndrehzahl := 1.400000e+03;
   Motordaten1.Nennstrom := 6.100000e+00;
   Motordaten1.Nennspannung := 2.310000e+02;
   Motordaten1.Nennleistung := 1.400000e+00;
   Motordaten2.Nennleistungsfaktor := 7.000000e-01;
   Motordaten2.Nennfrequenz := 1.000000e+02;
   Motordaten2.Nenndrehzahl := 2.000000e+02;
   Motordaten2.Nennstrom := 5.000000e+00;
   Motordaten2.Nennspannung := 3.800000e+02;
   Motordaten2.Nennleistung := 1.000000e+03;
   Motordaten3.Nennleistungsfaktor := 7.000000e-01;
   Motordaten3.Nennfrequenz := 1.000000e+02;
   Motordaten3.Nenndrehzahl := 2.000000e+02;
   Motordaten3.Nennstrom := 5.000000e+00;
   Motordaten3.Nennspannung := 3.800000e+02;
   Motordaten3.Nennleistung := 1.000000e+03;
   Motordaten4.Nennleistungsfaktor := 7.000000e-01;
   Motordaten4.Nennfrequenz := 1.000000e+02;
   Motordaten4.Nenndrehzahl := 2.000000e+02;
   Motordaten4.Nennstrom := 5.000000e+00;
   Motordaten4.Nennspannung := 3.800000e+02;
   Motordaten4.Nennleistung := 1.000000e+03;
   Motordaten5.Nennleistungsfaktor := 7.000000e-01;
   Motordaten5.Nennfrequenz := 1.000000e+02;
   Motordaten5.Nenndrehzahl := 2.000000e+02;
   Motordaten5.Nennstrom := 5.000000e+00;
   Motordaten5.Nennspannung := 3.800000e+02;
   Motordaten5.Nennleistung := 1.000000e+03;
   Motordaten6.Nennleistungsfaktor := 7.000000e-01;
   Motordaten6.Nennfrequenz := 1.000000e+02;
   Motordaten6.Nenndrehzahl := 2.000000e+02;
   Motordaten6.Nennstrom := 5.000000e+00;
   Motordaten6.Nennspannung := 3.800000e+02;
   Motordaten6.Nennleistung := 1.000000e+03;
   Motordaten7.Nennleistungsfaktor := 7.000000e-01;
   Motordaten7.Nennfrequenz := 1.000000e+02;
   Motordaten7.Nenndrehzahl := 2.000000e+02;
   Motordaten7.Nennstrom := 5.000000e+00;
   Motordaten7.Nennspannung := 3.800000e+02;
   Motordaten7.Nennleistung := 1.000000e+03;
   Motordaten8.Nennleistungsfaktor := 7.000000e-01;
   Motordaten8.Nennfrequenz := 1.000000e+02;
   Motordaten8.Nenndrehzahl := 2.000000e+02;
   Motordaten8.Nennstrom := 5.000000e+00;
   Motordaten8.Nennspannung := 3.800000e+02;
   Motordaten8.Nennleistung := 1.000000e+03;
   Motordaten9.Nennleistungsfaktor := 7.000000e-01;
   Motordaten9.Nennfrequenz := 1.000000e+02;
   Motordaten9.Nenndrehzahl := 2.000000e+02;
   Motordaten9.Nennstrom := 5.000000e+00;
   Motordaten9.Nennspannung := 3.800000e+02;
   Motordaten9.Nennleistung := 1.000000e+03;
   Motordaten10.Nennleistungsfaktor := 7.000000e-01;
   Motordaten10.Nennfrequenz := 1.000000e+02;
   Motordaten10.Nenndrehzahl := 2.000000e+02;
   Motordaten10.Nennstrom := 5.000000e+00;
   Motordaten10.Nennspannung := 3.800000e+02;
   Motordaten10.Nennleistung := 1.000000e+03;
END_DATA_BLOCK

DATA_BLOCK "DB30 Daten von/an FG"	// DB 30
AUTHOR : sra
FAMILY : hsh
VERSION : 0.0
"FB30 Daten von/an  FG"
BEGIN
END_DATA_BLOCK

DATA_BLOCK "DB32 Inputs"	// DB 32
AUTHOR : sra
FAMILY : SCADA
VERSION : 0.0
"FB32 Eingaege an FG"
BEGIN
END_DATA_BLOCK

DATA_BLOCK "DB33 Outputs"	// DB 33
AUTHOR : sra
FAMILY : SCADA
VERSION : 0.0
"FB33 Ausgaege an FG"
BEGIN
END_DATA_BLOCK

DATA_BLOCK "DB34 Faults"	// DB 34
AUTHOR : sra
FAMILY : AZO
VERSION : 0.0
"FB34 Störbearbeitung"
BEGIN
END_DATA_BLOCK

DATA_BLOCK "DB35 Acknolegments"	// DB 35
VERSION : 0.1
  STRUCT
   Quittierung : ARRAY  [0 .. 1023, 0 .. 7 ] OF BOOL  := FALSE;
   Quittierung_Spiegelungen : ARRAY  [0 .. 1023, 0 .. 7 ] OF BOOL  := FALSE;
  END_STRUCT ;	
BEGIN
END_DATA_BLOCK

DATA_BLOCK "DB92 Eingänge AVP"	// DB 92
VERSION : 0.0
"FB92 Eingänge AVP"
BEGIN
END_DATA_BLOCK

DATA_BLOCK "LINE1"	// DB 1000
AUTHOR : ilia
VERSION : 0.0
"****PRODUCTION****"
BEGIN
END_DATA_BLOCK

DATA_BLOCK "CONTAINERSTATION CST01"	// DB 1001
AUTHOR : ilia
VERSION : 0.1
"CONTAINERSTATION"
BEGIN
END_DATA_BLOCK

DATA_BLOCK "RECEIVER REC01"	// DB 1011
AUTHOR : ilia
VERSION : 0.1
"RECEIVER"
BEGIN
END_DATA_BLOCK

DATA_BLOCK "VP01"	// DB 1051
AUTHOR : ilia
VERSION : 0.1
"VACUUM PUMP"
BEGIN
END_DATA_BLOCK

DATA_BLOCK "RecipeData"	// DB 1111
VERSION : 0.1
  STRUCT
   RECIPE1 : STRUCT 	//Recipe
    RecipeName : STRING  [18 ] := 'RECIPE1';	//Recipe Name
    SpeedRinne : INT  := 30;	//Speed of Rinne
    SpeedRotaryFeeder : INT  := 30;	//Speed of RF
    SpeedVacuumPump : INT  := 35;	//Speed of VP1
    NumberOfPumps : INT  := 1;
    reserve1 : INT ;
    reserve2 : INT ;
    reserve3 : ARRAY  [1 .. 8 ] OF BYTE  := B#16#0;
   END_STRUCT ;
   RECIPE2 : STRUCT 	//Recipe
    RecipeName : STRING  [18 ] := 'RECIPE2';	//Recipe Name
    SpeedRinne : INT  := 30;	//Speed of Rinne
    SpeedRotaryFeeder : INT  := 30;	//Speed of RF
    SpeedVacuumPump : INT  := 35;	//Speed of VP1
    NumberOfPumps : INT  := 1;
    reserve1 : INT ;
    reserve2 : INT ;
    reserve3 : ARRAY  [1 .. 8 ] OF BYTE  := B#16#0;
   END_STRUCT ;
   RECIPE3 : STRUCT 	//Recipe
    RecipeName : STRING  [18 ] := 'RECIPE3';	//Recipe Name
    SpeedRinne : INT  := 30;	//Speed of Rinne
    SpeedRotaryFeeder : INT  := 30;	//Speed of RF
    SpeedVacuumPump : INT  := 35;	//Speed of VP1
    NumberOfPumps : INT  := 1;
    reserve1 : INT ;
    reserve2 : INT ;
    reserve3 : ARRAY  [1 .. 8 ] OF BYTE  := B#16#0;
   END_STRUCT ;
   RECIPE4 : STRUCT 	//Recipe
    RecipeName : STRING  [18 ] := 'RECIPE4';	//Recipe Name
    SpeedRinne : INT  := 30;	//Speed of Rinne
    SpeedRotaryFeeder : INT  := 30;	//Speed of RF
    SpeedVacuumPump : INT  := 35;	//Speed of VP1
    NumberOfPumps : INT  := 1;
    reserve1 : INT ;
    reserve2 : INT ;
    reserve3 : ARRAY  [1 .. 8 ] OF BYTE  := B#16#0;
   END_STRUCT ;
   RECIPE5 : STRUCT 	//Recipe
    RecipeName : STRING  [18 ] := 'RECIPE5';	//Recipe Name
    SpeedRinne : INT  := 30;	//Speed of Rinne
    SpeedRotaryFeeder : INT  := 30;	//Speed of RF
    SpeedVacuumPump : INT  := 35;	//Speed of VP1
    NumberOfPumps : INT  := 1;
    reserve1 : INT ;
    reserve2 : INT ;
    reserve3 : ARRAY  [1 .. 8 ] OF BYTE  := B#16#0;
   END_STRUCT ;
   RECIPE6 : STRUCT 	//Recipe
    RecipeName : STRING  [18 ] := 'RECIPE6';	//Recipe Name
    SpeedRinne : INT  := 30;	//Speed of Rinne
    SpeedRotaryFeeder : INT  := 30;	//Speed of RF
    SpeedVacuumPump : INT  := 35;	//Speed of VP1
    NumberOfPumps : INT  := 1;
    reserve1 : INT ;
    reserve2 : INT ;
    reserve3 : ARRAY  [1 .. 8 ] OF BYTE  := B#16#0;
   END_STRUCT ;
   RECIPE7 : STRUCT 	//Recipe
    RecipeName : STRING  [18 ] := 'RECIPE7';	//Recipe Name
    SpeedRinne : INT  := 30;	//Speed of Rinne
    SpeedRotaryFeeder : INT  := 30;	//Speed of RF
    SpeedVacuumPump : INT  := 35;	//Speed of VP1
    NumberOfPumps : INT  := 1;
    reserve1 : INT ;
    reserve2 : INT ;
    reserve3 : ARRAY  [1 .. 8 ] OF BYTE  := B#16#0;
   END_STRUCT ;
   RECIPE8 : STRUCT 	//Recipe
    RecipeName : STRING  [18 ] := 'RECIPE8';	//Recipe Name
    SpeedRinne : INT  := 30;	//Speed of Rinne
    SpeedRotaryFeeder : INT  := 30;	//Speed of RF
    SpeedVacuumPump : INT  := 35;	//Speed of VP1
    NumberOfPumps : INT  := 1;
    reserve1 : INT ;
    reserve2 : INT ;
    reserve3 : ARRAY  [1 .. 8 ] OF BYTE  := B#16#0;
   END_STRUCT ;
   RECIPE9 : STRUCT 	//Recipe
    RecipeName1 : STRING  [18 ] := 'RECIPE9';	//Recipe Name
    SpeedRinne : INT  := 30;	//Speed of Rinne
    SpeedRotaryFeeder : INT  := 30;	//Speed of RF
    SpeedVacuumPump : INT  := 35;	//Speed of VP1
    NumberOfPumps : INT  := 1;
    reserve1 : INT ;
    reserve2 : INT ;
    reserve3 : ARRAY  [1 .. 8 ] OF BYTE  := B#16#0;
   END_STRUCT ;
   RECIPE10 : STRUCT 	//Recipe
    RecipeName : STRING  [18 ] := 'RECIPE10';	//Recipe Name
    SpeedRinne : INT  := 30;	//Speed of Rinne
    SpeedRotaryFeeder : INT  := 30;	//Speed of RF
    SpeedVacuumPump : INT  := 35;	//Speed of VP1
    NumberOfPumps : INT  := 1;
    reserve1 : INT ;
    reserve2 : INT ;
    reserve3 : ARRAY  [1 .. 8 ] OF BYTE  := B#16#0;
   END_STRUCT ;
  END_STRUCT ;	
BEGIN
   RECIPE1.RecipeName := 'RECIPE1';
   RECIPE1.SpeedRinne := 30;
   RECIPE1.SpeedRotaryFeeder := 30;
   RECIPE1.SpeedVacuumPump := 35;
   RECIPE1.NumberOfPumps := 1;
   RECIPE2.RecipeName := 'RECIPE2';
   RECIPE2.SpeedRinne := 30;
   RECIPE2.SpeedRotaryFeeder := 30;
   RECIPE2.SpeedVacuumPump := 35;
   RECIPE2.NumberOfPumps := 1;
   RECIPE3.RecipeName := 'RECIPE3';
   RECIPE3.SpeedRinne := 30;
   RECIPE3.SpeedRotaryFeeder := 30;
   RECIPE3.SpeedVacuumPump := 35;
   RECIPE3.NumberOfPumps := 1;
   RECIPE4.RecipeName := 'RECIPE4';
   RECIPE4.SpeedRinne := 30;
   RECIPE4.SpeedRotaryFeeder := 30;
   RECIPE4.SpeedVacuumPump := 35;
   RECIPE4.NumberOfPumps := 1;
   RECIPE5.RecipeName := 'RECIPE5';
   RECIPE5.SpeedRinne := 30;
   RECIPE5.SpeedRotaryFeeder := 30;
   RECIPE5.SpeedVacuumPump := 35;
   RECIPE5.NumberOfPumps := 1;
   RECIPE6.RecipeName := 'RECIPE6';
   RECIPE6.SpeedRinne := 30;
   RECIPE6.SpeedRotaryFeeder := 30;
   RECIPE6.SpeedVacuumPump := 35;
   RECIPE6.NumberOfPumps := 1;
   RECIPE7.RecipeName := 'RECIPE7';
   RECIPE7.SpeedRinne := 30;
   RECIPE7.SpeedRotaryFeeder := 30;
   RECIPE7.SpeedVacuumPump := 35;
   RECIPE7.NumberOfPumps := 1;
   RECIPE8.RecipeName := 'RECIPE8';
   RECIPE8.SpeedRinne := 30;
   RECIPE8.SpeedRotaryFeeder := 30;
   RECIPE8.SpeedVacuumPump := 35;
   RECIPE8.NumberOfPumps := 1;
   RECIPE9.RecipeName1 := 'RECIPE9';
   RECIPE9.SpeedRinne := 30;
   RECIPE9.SpeedRotaryFeeder := 30;
   RECIPE9.SpeedVacuumPump := 35;
   RECIPE9.NumberOfPumps := 1;
   RECIPE10.RecipeName := 'RECIPE10';
   RECIPE10.SpeedRinne := 30;
   RECIPE10.SpeedRotaryFeeder := 30;
   RECIPE10.SpeedVacuumPump := 35;
   RECIPE10.NumberOfPumps := 1;
END_DATA_BLOCK

DATA_BLOCK "test"	// DB 2222
VERSION : 0.1
  STRUCT
   Recipe : STRUCT 	//Temporary placeholder variable
    Speed_1 : INT  := 1;
    Speed_2 : INT  := 2;
    Number : INT ;
   END_STRUCT ;
  END_STRUCT ;	
BEGIN
   Recipe.Speed_1 := 1;
   Recipe.Speed_2 := 2;
END_DATA_BLOCK

DATA_BLOCK "FREQUENCY CONVERTERS"	// DB 4900
AUTHOR : ilia
VERSION : 0.0
"*** FCs ***"
BEGIN
END_DATA_BLOCK

DATA_BLOCK "FC VACUUM PUMP"	// DB 10001
VERSION : 0.0
"FREQ.CONVERTER"
BEGIN
END_DATA_BLOCK

DATA_BLOCK "FC ROTARY FEEDER REC01"	// DB 10002
VERSION : 0.0
"FREQ.CONVERTER"
BEGIN
END_DATA_BLOCK

ORGANIZATION_BLOCK "OB 1 Zyklisches Prg."	// OB 1
TITLE = zyklischer Programmablauf
//Erstellung:
//Datum        Bearbeiter                                                 Version
//--------------------------------------------------------------------------------
//01.08.18     Ilia Bedniakov                                             01.00.00
//
//Änderungen:
//Nr. Datum    Bearb Beschreibung                                   Marke Version
//--------------------------------------------------------------------------------
//01  
//
VERSION : 0.1
VAR_TEMP
  OB1_EV_CLASS : BYTE ;	//Bits 0-3 = 1 (Coming event), Bits 4-7 = 1 (Event class 1)
  OB1_SCAN_1 : BYTE ;	//1 (Cold restart scan 1 of OB 1), 3 (Scan 2-n of OB 1)
  OB1_PRIORITY : BYTE ;	//1 (Priority of 1 is lowest)
  OB1_OB_NUMBR : BYTE ;	//1 (Organization block 1, OB1)
  OB1_RESERVED_1 : BYTE ;	//Reserved for system
  OB1_RESERVED_2 : BYTE ;	//Reserved for system
  OB1_PREV_CYCLE : INT ;	//Cycle time of previous OB1 scan (milliseconds)
  OB1_MIN_CYCLE : INT ;	//Minimum cycle time of OB1 (milliseconds)
  OB1_MAX_CYCLE : INT ;	//Maximum cycle time of OB1 (milliseconds)
  OB1_DATE_TIME : DATE_AND_TIME ;	//Date and time OB1 started
  DUMMY_INT : INT ;
  dummybool : BOOL ;
END_VAR
BEGIN
NETWORK
TITLE = Simulation
//      CLR   
      SET;
      =     "M0.5 SimulationInternal";
      A     "M0.5 SimulationInternal";
      JCN   NS;	// No simulation
      CALL  "CMs_SIMULATION" , "CMs_SIMULATION_DB";
NS:   NOP   0;
NETWORK
TITLE = Datum, Uhrzeit und Zykluszeiten in DB3 kopieren
      CALL  "BLKMOV" (
           SRCBLK                   := #OB1_DATE_TIME,
           RET_VAL                  := #DUMMY_INT,
           DSTBLK                   := "DB3 CPU Daten".OB1_Info.OB1_DATE_TIME);
      L     #OB1_PREV_CYCLE;
      T     "DB3 CPU Daten".OB1_Info.OB1_PREV_CYCLE;
      L     #OB1_MIN_CYCLE;
      T     "DB3 CPU Daten".OB1_Info.OB1_MIN_CYCLE;
      L     #OB1_MAX_CYCLE;
      T     "DB3 CPU Daten".OB1_Info.OB1_MAX_CYCLE;
NETWORK
TITLE = Standardsignale
      CALL  "FC13 Standardsignale" (
           in_E_Sicherung_OK        := "01_01_101_Gn",
           in_Basistakt_Timer       := "M4.1 ImpulseClock0,2Sec",
           in_Zeit_Basistakt_100ms  := 2,
           o_Lampe_Stoer_Sicherung  := #dummybool,
           o_Stoerung_Sicherung     := #dummybool);
NETWORK
TITLE = Daten von/an HMI
      CALL  "FB30 Daten von/an  FG" , "DB30 Daten von/an FG";
      CALL  "FB32 Eingaege an FG" , "DB32 Inputs";
      CALL  "FB33 Ausgaege an FG" , "DB33 Outputs";
NETWORK
TITLE = Stoerungen Auswertung
      CALL  "FB34 Störbearbeitung" , "DB34 Faults";
NETWORK
TITLE = Anwenderprogramm
      CALL  "****PRODUCTION****" , "LINE1";
NETWORK
TITLE = Neustart oder Wiederanlauf SPS rücksetzen
//letztes Netzwerk
      SET;
      R     "M1.3 CompleteRestart";
      R     "M1.4 RestartPLC";
END_ORGANIZATION_BLOCK

ORGANIZATION_BLOCK "OB 80 Zeitfehler-OB"	// OB 80
TITLE = Zeitfehler
//Erstellung:
//Datum        Bearbeiter                                                 Version
//--------------------------------------------------------------------------------
//03.06.98     Rainer Schaffert (sra)                                     01.00.00
//
//Änderungen:
//Nr. Datum    Bearb Beschreibung                                   Marke Version
//--------------------------------------------------------------------------------
//01  
//
//________________________________________________________________________________
//OB wird bei Zeitfehler bearbeitet
//
AUTHOR : sra
FAMILY : error_OB
NAME : time_err
VERSION : 0.1
VAR_TEMP
  OB80_EV_CLASS : BYTE ;	//16#35, Event class 3, Entering event state, Internal fault event
  OB80_FLT_ID : BYTE ;	//16#XX, Fault identifcation code
  OB80_PRIORITY : BYTE ;	//26 (Priority of 1 is lowest)
  OB80_OB_NUMBR : BYTE ;	//80 (Organization block 80, OB80)
  OB80_RESERVED_1 : BYTE ;	//Reserved for system
  OB80_RESERVED_2 : BYTE ;	//Reserved for system
  OB80_ERROR_INFO : WORD ;	//Error information on event
  OB80_ERR_EV_CLASS : BYTE ;	//Class of event causing error
  OB80_ERR_EV_NUM : BYTE ;	//Number of event causing error
  OB80_OB_PRIORITY : BYTE ;	//Priority of OB causing error
  OB80_OB_NUM : BYTE ;	//Number of OB causing error
  OB80_DATE_TIME : DATE_AND_TIME ;	//Date and time OB80 started
END_VAR
BEGIN
NETWORK
TITLE = Fehlermeldung erzeugen
//Fehlermeldung erzeugen
//
//Fehlercode B#16#01 : Zykluszeit überschritten
//                     OB80_ERROR_INFO: Laufzeit des letzten Zyklus
//           
//           B#16#02 : Der angeforderte OB ist noch in Bearbeitung
//
//           B#16#07 : Überlauf des OB-Anforderungspuffers für die aktuelle 
//                     Prioritätsklasse
//
//           B#16#05 : abgelaufener Urzeitalarm durch Urzeitsprung
//
//           B#16#06 : abgelaufener Urzeitalarm bei Wiedereintritt 
//
      L     #OB80_FLT_ID;
      L     B#16#0;
      <>I;
      =     "DB3 CPU Daten".Fehler_OB_Info.Zeitfehler_OB80;
      L     #OB80_FLT_ID;
      T     "DB3 CPU Daten".Fehler_OB_Info.OB_80_Fault_ID;
END_ORGANIZATION_BLOCK

ORGANIZATION_BLOCK "OB 82 Diagnosealarm-OB"	// OB 82
TITLE = Diagnose-Alarm
//Erstellung:
//Datum        Bearbeiter                                                 Version
//--------------------------------------------------------------------------------
//03.06.98     Rainer Schaffert (sra)                                     01.00.00
//
//Änderungen:
//Nr. Datum    Bearb Beschreibung                                   Marke Version
//--------------------------------------------------------------------------------
//01  
//
//________________________________________________________________________________
//OB wird bei Diagnose-Alarm bearbeitet
//
AUTHOR : sra
FAMILY : error_OB
NAME : diagn_OB
VERSION : 0.1
VAR_TEMP
  OB82_EV_CLASS : BYTE ;	//16#39, Event class 3, Entering event state, Internal fault event
  OB82_FLT_ID : BYTE ;	//16#XX, Fault identifcation code
  OB82_PRIORITY : BYTE ;	//26/28 (Priority of 1 is lowest)
  OB82_OB_NUMBR : BYTE ;	//82 (Organization block 82, OB82)
  OB82_RESERVED_1 : BYTE ;	//Reserved for system
  OB82_IO_FLAG : BYTE ;	//Input (01010100), Output (01010101)
  OB82_MDL_ADDR : INT ;	//Base address of module with fault
  OB82_MDL_DEFECT : BOOL ;	//Module defective
  OB82_INT_FAULT : BOOL ;	//Internal fault
  OB82_EXT_FAULT : BOOL ;	//External fault
  OB82_PNT_INFO : BOOL ;	//Point information
  OB82_EXT_VOLTAGE : BOOL ;	//External voltage low
  OB82_FLD_CONNCTR : BOOL ;	//Field wiring connector missing
  OB82_NO_CONFIG : BOOL ;	//Module has no configuration data
  OB82_CONFIG_ERR : BOOL ;	//Module has configuration error
  OB82_MDL_TYPE : BYTE ;	//Type of module
  OB82_SUB_NDL_ERR : BOOL ;	//Sub-Module is missing or has error
  OB82_COMM_FAULT : BOOL ;	//Communication fault
  OB82_MDL_STOP : BOOL ;	//Module is stopped
  OB82_WTCH_DOG_FLT : BOOL ;	//Watch dog timer stopped module
  OB82_INT_PS_FLT : BOOL ;	//Internal power supply fault
  OB82_PRIM_BATT_FLT : BOOL ;	//Primary battery is in fault
  OB82_BCKUP_BATT_FLT : BOOL ;	//Backup battery is in fault
  OB82_RESERVED_2 : BOOL ;	//Reserved for system
  OB82_RACK_FLT : BOOL ;	//Rack fault, only for bus interface module
  OB82_PROC_FLT : BOOL ;	//Processor fault
  OB82_EPROM_FLT : BOOL ;	//EPROM fault
  OB82_RAM_FLT : BOOL ;	//RAM fault
  OB82_ADU_FLT : BOOL ;	//ADU fault
  OB82_FUSE_FLT : BOOL ;	//Fuse fault
  OB82_HW_INTR_FLT : BOOL ;	//Hardware interupt input in fault
  OB82_RESERVED_3 : BOOL ;	//Reserved for system
  OB82_DATE_TIME : DATE_AND_TIME ;	//Date and time OB82 started
END_VAR
BEGIN
NETWORK
TITLE = Fehlermeldung erzeugen
//Fehlermeldung erzeugen
//
//Fehlercode B#16#42 : 
//
      A(;
      L     #OB82_EV_CLASS;
      L     B#16#39;	// kommendes Ereignis
      ==I;
      );
      A(;
      L     #OB82_FLT_ID;
      L     B#16#0;
      <>I;
      );
      =     "DB3 CPU Daten".Fehler_OB_Info.Diagnose_Alarm_OB82;
      L     #OB82_FLT_ID;
      T     "DB3 CPU Daten".Fehler_OB_Info.OB_82_Fault_ID;
END_ORGANIZATION_BLOCK

ORGANIZATION_BLOCK "OB 83 Ziehen-/Stecken-OB"	// OB 83
TITLE = Ziehen/Stecken-Alarm
//Erstellung:
//Datum        Bearbeiter                                                 Version
//--------------------------------------------------------------------------------
//03.06.98     Rainer Schaffert (sra)                                     01.00.00
//
//Änderungen:
//Nr. Datum    Bearb Beschreibung                                   Marke Version
//--------------------------------------------------------------------------------
//01  
//
//________________________________________________________________________________
//OB wird bei Ziehen/Stecken-Alarm bearbeitet
//
AUTHOR : sra
FAMILY : AZO
VERSION : 0.0
VAR_TEMP
  OB83_EV_CLASS : BYTE ;	//16#38/39, Event class 3, module inserted/removed (8/9)
  OB83_FLT_ID : BYTE ;	//16#XX, Fault identifcation code
  OB83_PRIORITY : BYTE ;	//26/28 (Priority of 1 is lowest)
  OB83_OB_NUMBR : BYTE ;	//83 (Organization block 83, OB83)
  OB83_RESERVED_1 : BYTE ;	//Reserved for system
  OB83_MDL_ID : BYTE ;	//Input module (01010100), Output module (01010101)
  OB83_MDL_ADDR : WORD ;	//Base address of module with point fault
  OB83_RACK_NUM : WORD ;	//Number of rack that has module with point fault
  OB83_MDL_TYPE : WORD ;	//Module type with point fault
  OB83_DATE_TIME : DATE_AND_TIME ;	//Date and time OB83 started
END_VAR
BEGIN
NETWORK
TITLE = Fehlermeldung erzeugen
//Fehlermeldung erzeugen
//
//Fehlercode B#16#61 : Baugruppe gezogen bzw. nicht ansprechbar (bei 
//                     Ereignisklasse B#16#39)
//                     Baugruppe gesteckt, Baugruppentyp ok (bei
//                     Ereignisklasse B#16#38)
//           
//           B#16#63 : Baugruppe gesteckt, jedoch falscher Baugruppentyp
//
//           B#16#64 : Baugruppe gesteckt, jedoch gestört(Typkennung nicht lesbar)
//
      A(;
      L     #OB83_EV_CLASS;
      L     B#16#39;	// kommendes Ereignis
      ==I;
      );
      A(;
      L     #OB83_FLT_ID;
      L     B#16#0;
      <>I;
      );
      =     "DB3 CPU Daten".Fehler_OB_Info.Ziehen_Stecken_OB83;
      L     #OB83_FLT_ID;
      T     "DB3 CPU Daten".Fehler_OB_Info.OB_83_Fault_ID;
END_ORGANIZATION_BLOCK

ORGANIZATION_BLOCK "OB 85 Prgablauffehler-OB"	// OB 85
TITLE = Programmablauffehler
//Erstellung:
//Datum        Bearbeiter                                                 Version
//--------------------------------------------------------------------------------
//03.06.98     Rainer Schaffert (sra)                                     01.00.00
//
//Änderungen:
//Nr. Datum    Bearb Beschreibung                                   Marke Version
//--------------------------------------------------------------------------------
//01  
//
//________________________________________________________________________________
//OB wird bei Programmablauffehler bearbeitet
//
//
AUTHOR : sra
FAMILY : AZO
VERSION : 0.0
VAR_TEMP
  OB85_EV_CLASS : BYTE ;	//16#35 Event class 3
  OB85_FLT_ID : BYTE ;	//16#XX, Fault identification code
  OB85_PRIORITY : BYTE ;	//26 (Priority of 1 is lowest)
  OB85_OB_NUMBR : BYTE ;	//85 (Organization block 85, OB85)
  OB85_RESERVED_1 : BYTE ;	//Reserved for system
  OB85_RESERVED_2 : BYTE ;	//Reserved for system
  OB85_RESERVED_3 : INT ;	//Reserved for system
  OB85_ERR_EV_CLASS : BYTE ;	//Class of event causing error
  OB85_ERR_EV_NUM : BYTE ;	//Number of event causing error
  OB85_OB_PRIOR : BYTE ;	//Priority of OB causing error
  OB85_OB_NUM : BYTE ;	//Number of OB causing error
  OB85_DATE_TIME : DATE_AND_TIME ;	//Date and time OB85 started
END_VAR
BEGIN
NETWORK
TITLE = Fehlermeldung erzeugen
//Fehlermeldung erzeugen
//
//Fehlercode B#16#A1 : Das Programm oder das Betriebssystem erzeugt ein 
//                     Startereignis für einen OB, der nicht in die CPU geladen 
//                     ist.
//
//           B#16#A2 : Das Programm oder das Betriebssystem erzeugt ein 
//                     Startereignis für einen OB, der nicht in die CPU geladen 
//                     ist.
//
//           B#16#A3 : Fehler beim Zugriff des Betriebssystems auf einen Baustein
//
//           B#16#B1 : Peripheriezugriffsfehler beim Aktualisieren des 
//                     Gesamtprozessabbildes der Eingänge
//
//           B#16#B1 : Peripheriezugriffsfehler beim Aktualisieren des            
//                     Gesamtprozessabbildes der Ausgänge
//
      L     #OB85_FLT_ID;
      L     B#16#0;
      <>I;
      =     "DB3 CPU Daten".Fehler_OB_Info.Programmablauf_OB85;
      L     #OB85_FLT_ID;
      T     "DB3 CPU Daten".Fehler_OB_Info.OB_85_Fault_ID;
END_ORGANIZATION_BLOCK

ORGANIZATION_BLOCK "OB 86 Baugr träger-OB"	// OB 86
TITLE = Baugruppenträgerausfall
//Erstellung:
//Datum        Bearbeiter                                                 Version
//--------------------------------------------------------------------------------
//03.06.98     Rainer Schaffert (sra)                                     01.00.00
//
//Änderungen:
//Nr. Datum    Bearb Beschreibung                                   Marke Version
//--------------------------------------------------------------------------------
//01  
//
//________________________________________________________________________________
//OB wird bei Baugruppenträgerausfall bearbeitet
//
AUTHOR : sra
FAMILY : AZO
VERSION : 0.0
VAR_TEMP
  OB86_EV_CLASS : BYTE ;	//16#38/39 Event class 3
  OB86_FLT_ID : BYTE ;	//16#C1/C4/C5, Fault identification code
  OB86_PRIORITY : BYTE ;	//26/28 (Priority of 1 is lowest)
  OB86_OB_NUMBR : BYTE ;	//86 (Organization block 86, OB86)
  OB86_RESERVED_1 : BYTE ;	//Reserved for system
  OB86_RESERVED_2 : BYTE ;	//Reserved for system
  OB86_MDL_ADDR : WORD ;	//Depending on fault identification code
  OB86_RACKS_FLTD : ARRAY  [0 .. 31 ] OF BOOL ;	//Racks in fault
  OB86_DATE_TIME : DATE_AND_TIME ;	//Date and time OB86 started
END_VAR
BEGIN
NETWORK
TITLE = Fehlermeldung erzeugen
//Fehlermeldung erzeugen
//
//Fehlercode B#16#C1 : Baugruppenträgerausfall
//
//           B#16#C2 : Baugruppenträgerwiederkehr (Baugruppenträgerausfall gehend 
//                     mit Abweichung Soll-/Istausbau)
//
//           B#16#C3 : Dezentrale Peripherie: Ausfall eines DP-Mastersystems
//
//           B#16#C4 : Ausfall einer DP-Station
//
//           B#16#C5 : Störung einer DP-Station
//
      A(;
      L     #OB86_EV_CLASS;
      L     B#16#39;	// kommendes Ereignis
      ==I;
      );
      A(;
      L     #OB86_FLT_ID;
      L     B#16#0;
      <>I;
      );
      =     "DB3 CPU Daten".Fehler_OB_Info.Baugr_tr_ausfall_OB86;
      L     #OB86_FLT_ID;
      T     "DB3 CPU Daten".Fehler_OB_Info.OB_86_Fault_ID;
END_ORGANIZATION_BLOCK

ORGANIZATION_BLOCK "OB 87 Kommunikations-OB"	// OB 87
TITLE = Kommunikationsfehler
//Erstellung:
//Datum        Bearbeiter                                                 Version
//--------------------------------------------------------------------------------
//03.06.98     Rainer Schaffert (sra)                                     01.00.00
//
//Änderungen:
//Nr. Datum    Bearb Beschreibung                                   Marke Version
//--------------------------------------------------------------------------------
//01  
//
//________________________________________________________________________________
//OB wird bei Kommunikationsfehler bearbeitet
//
AUTHOR : sra
FAMILY : AZO
VERSION : 0.0
VAR_TEMP
  OB87_EV_CLASS : BYTE ;	//16#35 Event class 3
  OB87_FLT_ID : BYTE ;	//16#XX, Fault identifcation code
  OB87_PRIORITY : BYTE ;	//26 (Priority of 1 is lowest)
  OB87_OB_NUMBR : BYTE ;	//87 (Organization block 87, OB87)
  OB87_RESERVED_1 : BYTE ;	//Reserved for system
  OB87_RESERVED_2 : BYTE ;	//Reserved for system
  OB87_RESERVED_3 : WORD ;	//Reserved for system
  OB87_RESERVED_4 : DWORD ;	//Reserved for system
  OB87_DATE_TIME : DATE_AND_TIME ;	//Date and time OB87 started
END_VAR
BEGIN
NETWORK
TITLE = Fehlermeldung erzeugen
//Fehlermeldung erzeugen
//
//Fehlercode B#16#D2 : Senden der Diagnoseeinträge nicht möglich
//
//           B#16#D3 : Synchronisationsdiagramme können nicht gesendet werden
//
//           B#16#D4 : Unzulässiger Uhrzeitsprung durch Uhrzeitsynchronisation
//
//           B#16#D5 : Fehler bei Übernahme der Synchronisationszeit
//
//           B#16#E1 : Falsche Telegrammkennung bei Globaldatenkommunikation
//
//           B#16#E3 : Telegrammlängenfehler bei Globaldatenkommunikation
//
//           B#16#E4 : Unzulässige GD-Paketnummer empfangen
//
//           B#16#E2 : GD-Paketstatus ist nicht in einen DP-eintragbar
//
//           B#16#E5 : Fehler bei Zugriff auf DB beim Datenaustausch über 
//                     Kommunikationsfunktionsbausteine
//
//           B#16#E6 : GD-Gesamtstatus ist nicht in DB eintragbar
//
      L     #OB87_FLT_ID;
      L     B#16#0;
      <>I;
      =     "DB3 CPU Daten".Fehler_OB_Info.Kommunikation_OB87;
      L     #OB87_FLT_ID;
      T     "DB3 CPU Daten".Fehler_OB_Info.OB_87_Fault_ID;
END_ORGANIZATION_BLOCK

ORGANIZATION_BLOCK "OB 100 Neustart-OB"	// OB 100
TITLE = Neustart
//Erstellung:
//Datum        Bearbeiter                                                 Version
//--------------------------------------------------------------------------------
//04.09.2001   R.Schaffert (sra)                                          01.00.00
//  
//Änderungen:
//Nr. Datum    Bearb Änderung                                       Marke  Version
//--------------------------------------------------------------------------------
//01  24.04.17 gea  set service mode lock auto                      (001) 01.00.01
//________________________________________________________________________________
//Programm wird am Anfang von OB 1 fortgesetzt
AUTHOR : sra
FAMILY : AZO
VERSION : 0.0
VAR_TEMP
  OB100_EV_CLASS : BYTE ;	//16#13, Event class 1, Entering event state, Event logged in diagnostic buffer
  OB100_STRTUP : BYTE ;	//16#81/82/83/84 Method of startup
  OB100_PRIORITY : BYTE ;	//27 (Priority of 1 is lowest)
  OB100_OB_NUMBR : BYTE ;	//100 (Organization block 100, OB100)
  OB100_RESERVED_1 : BYTE ;	//Reserved for system
  OB100_RESERVED_2 : BYTE ;	//Reserved for system
  OB100_STOP : WORD ;	//Event that caused CPU to stop (16#4xxx)
  OB100_STRT_INFO : DWORD ;	//Information on how system started
  OB100_DATE_TIME : DATE_AND_TIME ;	//Date and time OB100 started
END_VAR
BEGIN
NETWORK
TITLE = Neustartmerker setzen
      SET;
      S     "M1.3 CompleteRestart";
      SET;	// (001)
      S     "Service Mode ExpertMode";	// (001)
END_ORGANIZATION_BLOCK

ORGANIZATION_BLOCK "OB 121 Programmierf-OB"	// OB 121
TITLE = Programmierfehler-OB
//Erstellung:
//Datum        Bearbeiter                                                 Version
//--------------------------------------------------------------------------------
//03.06.98     Rainer Schaffert (sra)                                     01.00.00
//
//Änderungen:
//Nr. Datum    Bearb Beschreibung                                   Marke Version
//--------------------------------------------------------------------------------
//01  
//
//________________________________________________________________________________
//OB wird aufgerufen wenn ein Fehler während der Programmbearbeitung auftritt
AUTHOR : sra
FAMILY : AZO
VERSION : 0.0
VAR_TEMP
  OB121_EV_CLASS : BYTE ;	//16#25, Event class 2, Entering event state, Internal fault event
  OB121_SW_FLT : BYTE ;	//16#XX Software programming fault
  OB121_PRIORITY : BYTE ;	//X = Priority of OB where fault occured (Priority of 1 is lowest)
  OB121_OB_NUMBR : BYTE ;	//121 (Organization block 121, OB121)
  OB121_BLK_TYPE : BYTE ;	//16#88/8A/8B/8C/8E Type of block fault occured in
  OB121_RESERVED_1 : BYTE ;	//Reserved for system
  OB121_FLT_REG : WORD ;	//16#XX Specific register that caused fault
  OB121_BLK_NUM : WORD ;	//Number of block that programming fault occured in
  OB121_PRG_ADDR : WORD ;	//Address in block where programming fault occured
  OB121_DATE_TIME : DATE_AND_TIME ;	//Date and time OB121 started
END_VAR
BEGIN
NETWORK
TITLE = Fehlermeldung erzeugen
//Fehlermeldung erzeugen
//
//Fehlercode B#16#21 : BCD-Konvertierungsfehler
//                                
//           B#16#22 : Bereichslängenfehler bei lesen
//
//           B#16#23 : Bereichslängenfehler bei schreiben
//
//           B#16#28 : lesender Zugriff auf ein Byte, Wort oder Doppelwort mit 
//                     einem Pointer, dessen Bitadresse ungleich 0 ist.
//
//           B#16#29 : schreibender Zugriff auf ein Byte, Wort oder Doppelwort 
//                     mit einem Pointer, dessen Bitadresse ungleich 0 ist.
//
//           B#16#24 : Bereichsfehler bei lesen
//
//           B#16#25 : Bereichsfehler bei schreiben
//
//           B#16#26 : Fehler bei Timernummer
//
//           B#16#27 : Fehler bei Zählernummer
//
//           B#16#30 : Schreibender Zugriff auf einen schreibgeschützten Global-DB
//
//           B#16#31 : Schreibender Zugriff auf einen schreibgeschützten 
//                     Instanz-DB
//
//           B#16#32 : DB-Nummernfehler beim Zugriff auf einen Global-DB
//
//           B#16#33 : DB-Nummernfehler beim Zugriff auf einen Instanz-DB
//
//
//
//Fehlermeldung erzeugen
//
//Fehlercode B#16#21 : BCD-Konvertierungsfehler
//                                
//           B#16#22 : Bereichslängenfehler bei lesen
//
//           B#16#23 : Bereichslängenfehler bei schreiben
//
//           B#16#28 : lesender Zugriff auf ein Byte, Wort oder Doppelwort mit 
//                     einem Pointer, dessen Bitadresse ungleich 0 ist.
//
//           B#16#29 : schreibender Zugriff auf ein Byte, Wort oder Doppelwort 
//mit 
//                     einem Pointer, dessen Bitadresse ungleich 0 ist.
//
//           B#16#24 : Bereichsfehler bei lesen
//
//           B#16#25 : Bereichsfehler bei schreiben
//
//           B#16#26 : Fehler bei Timernummer
//
//           B#16#27 : Fehler bei Zählernummer
//
//           B#16#30 : Schreibender Zugriff auf einen schreibgeschützten Global-DB
//
//           B#16#31 : Schreibender Zugriff auf einen schreibgeschützten 
//                     Instanz-DB
//
//           B#16#32 : DB-Nummernfehler beim Zugriff auf einen Global-DB
//
//           B#16#33 : DB-Nummernfehler beim Zugriff auf einen Instanz-DB
//
//           B#16#34 : FC-Nummernfehler beim FC-Aufruf
//
//           B#16#35 : FB-Nummernfehler beim FB-Aufruf
//
//           B#16#3A : Zugriff auf einen nicht geladenen DB
//
//           B#16#3C : Zugriff auf einen nicht geladenen FC
//
//           B#16#3D : Zugriff auf einen nicht geladenen SFC
//
//           B#16#3E : Zugriff auf einen nicht geladenen FB
//
//           B#16#3F : Zugriff auf einen nicht geladenen SFB
//
//
      A(;
      L     #OB121_SW_FLT;
      L     B#16#0;
      <>I;
      );
      =     "DB3 CPU Daten".Fehler_OB_Info.Programmierfehler_OB121;
      L     #OB121_SW_FLT;
      T     "DB3 CPU Daten".Fehler_OB_Info.OB_121_Fault_ID;
END_ORGANIZATION_BLOCK
